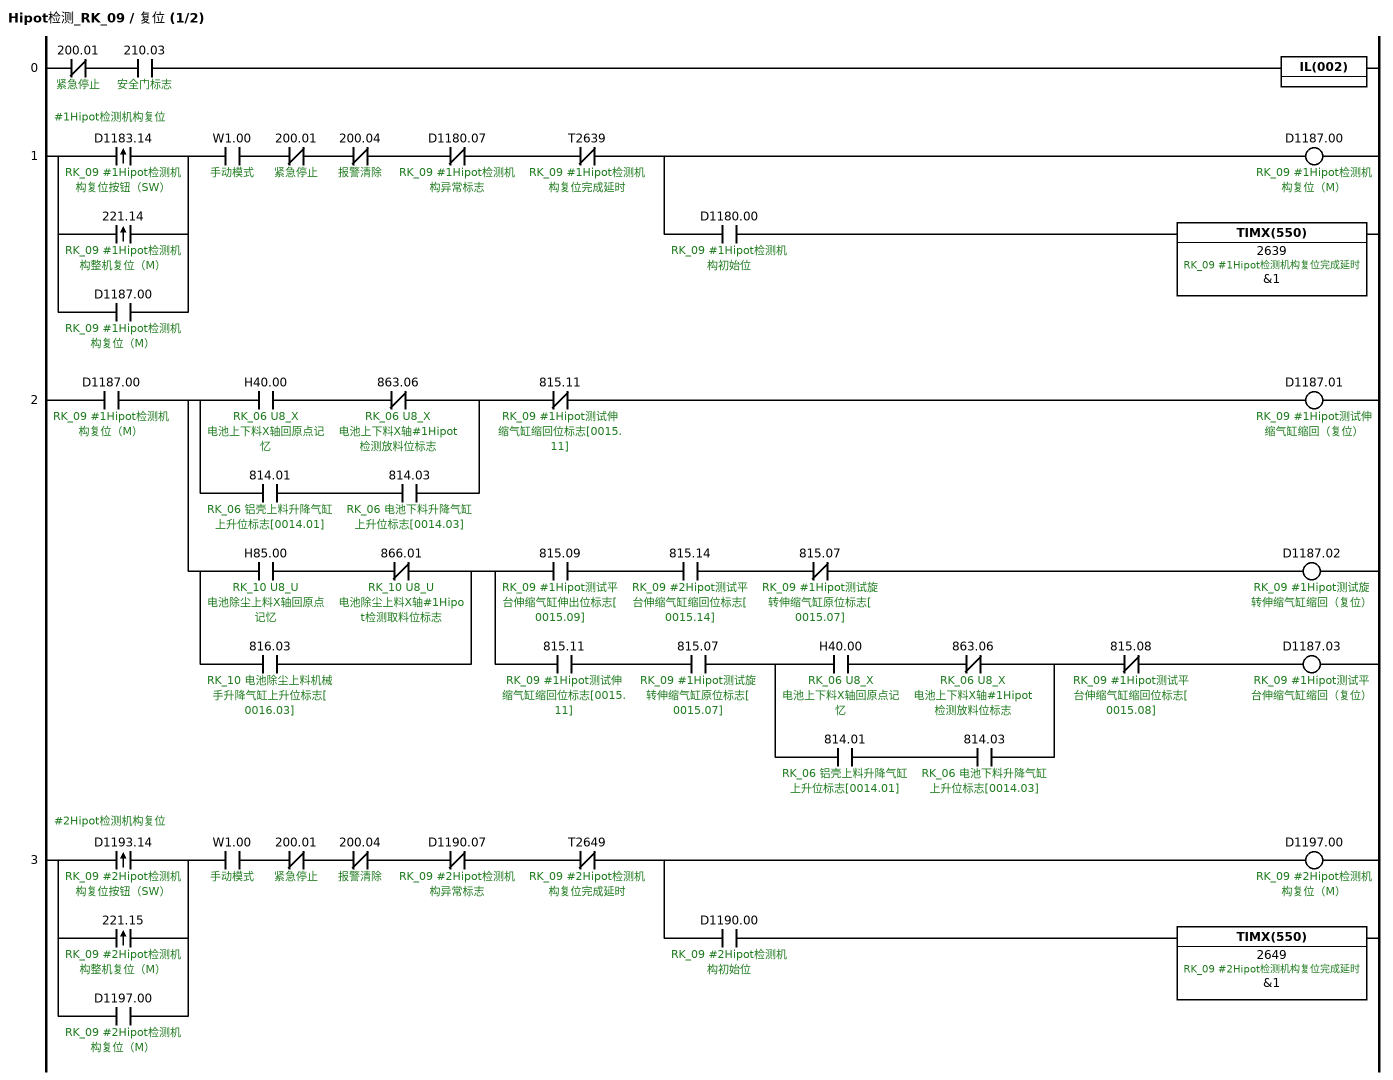
; [picture p672: Hipot检测_RK_09 / 复位, rungs 0-3]
; rung 0
LDNOT 200.01  ; 紧急停止
AND 210.03  ; 安全门标志
IL(002)
; rung 1: #1Hipot检测机构复位
@LD D1183.14  ; RK_09 #1Hipot检测机构复位按钮（SW）
@OR 221.14  ; RK_09 #1Hipot检测机构整机复位（M）
OR D1187.00  ; RK_09 #1Hipot检测机构复位（M）
AND W1.00  ; 手动模式
ANDNOT 200.01  ; 紧急停止
ANDNOT 200.04  ; 报警清除
ANDNOT D1180.07  ; RK_09 #1Hipot检测机构异常标志
ANDNOT T2639  ; RK_09 #1Hipot检测机构复位完成延时
OUT D1187.00  ; RK_09 #1Hipot检测机构复位（M）
AND D1180.00  ; RK_09 #1Hipot检测机构初始位
TIMX(550) 2639 &1  ; RK_09 #1Hipot检测机构复位完成延时
; rung 2
LD D1187.00  ; RK_09 #1Hipot检测机构复位（M）
OUT TR0
LD H40.00  ; RK_06 U8_X 电池上下料X轴回原点记忆
ANDNOT 863.06  ; RK_06 U8_X 电池上下料X轴#1Hipot检测放料位标志
LD 814.01  ; RK_06 铝壳上料升降气缸上升位标志[0014.01]
AND 814.03  ; RK_06 电池下料升降气缸上升位标志[0014.03]
ORLD
ANDLD
ANDNOT 815.11  ; RK_09 #1Hipot测试伸缩气缸缩回位标志[0015.11]
OUT D1187.01  ; RK_09 #1Hipot测试伸缩气缸缩回（复位）
LD TR0
LD H85.00  ; RK_10 U8_U 电池除尘上料X轴回原点记忆
ANDNOT 866.01  ; RK_10 U8_U 电池除尘上料X轴#1Hipot检测取料位标志
OR 816.03  ; RK_10 电池除尘上料机械手升降气缸上升位标志[0016.03]
ANDLD
OUT TR0
AND 815.09  ; RK_09 #1Hipot测试平台伸缩气缸伸出位标志[0015.09]
AND 815.14  ; RK_09 #2Hipot测试平台伸缩气缸缩回位标志[0015.14]
ANDNOT 815.07  ; RK_09 #1Hipot测试旋转伸缩气缸原位标志[0015.07]
OUT D1187.02  ; RK_09 #1Hipot测试旋转伸缩气缸缩回（复位）
LD TR0
AND 815.11  ; RK_09 #1Hipot测试伸缩气缸缩回位标志[0015.11]
AND 815.07  ; RK_09 #1Hipot测试旋转伸缩气缸原位标志[0015.07]
LD H40.00  ; RK_06 U8_X 电池上下料X轴回原点记忆
ANDNOT 863.06  ; RK_06 U8_X 电池上下料X轴#1Hipot检测放料位标志
LD 814.01  ; RK_06 铝壳上料升降气缸上升位标志[0014.01]
AND 814.03  ; RK_06 电池下料升降气缸上升位标志[0014.03]
ORLD
ANDLD
ANDNOT 815.08  ; RK_09 #1Hipot测试平台伸缩气缸缩回位标志[0015.08]
OUT D1187.03  ; RK_09 #1Hipot测试平台伸缩气缸缩回（复位）
; rung 3: #2Hipot检测机构复位
@LD D1193.14  ; RK_09 #2Hipot检测机构复位按钮（SW）
@OR 221.15  ; RK_09 #2Hipot检测机构整机复位（M）
OR D1197.00  ; RK_09 #2Hipot检测机构复位（M）
AND W1.00  ; 手动模式
ANDNOT 200.01  ; 紧急停止
ANDNOT 200.04  ; 报警清除
ANDNOT D1190.07  ; RK_09 #2Hipot检测机构异常标志
ANDNOT T2649  ; RK_09 #2Hipot检测机构复位完成延时
OUT D1197.00  ; RK_09 #2Hipot检测机构复位（M）
AND D1190.00  ; RK_09 #2Hipot检测机构初始位
TIMX(550) 2649 &1  ; RK_09 #2Hipot检测机构复位完成延时

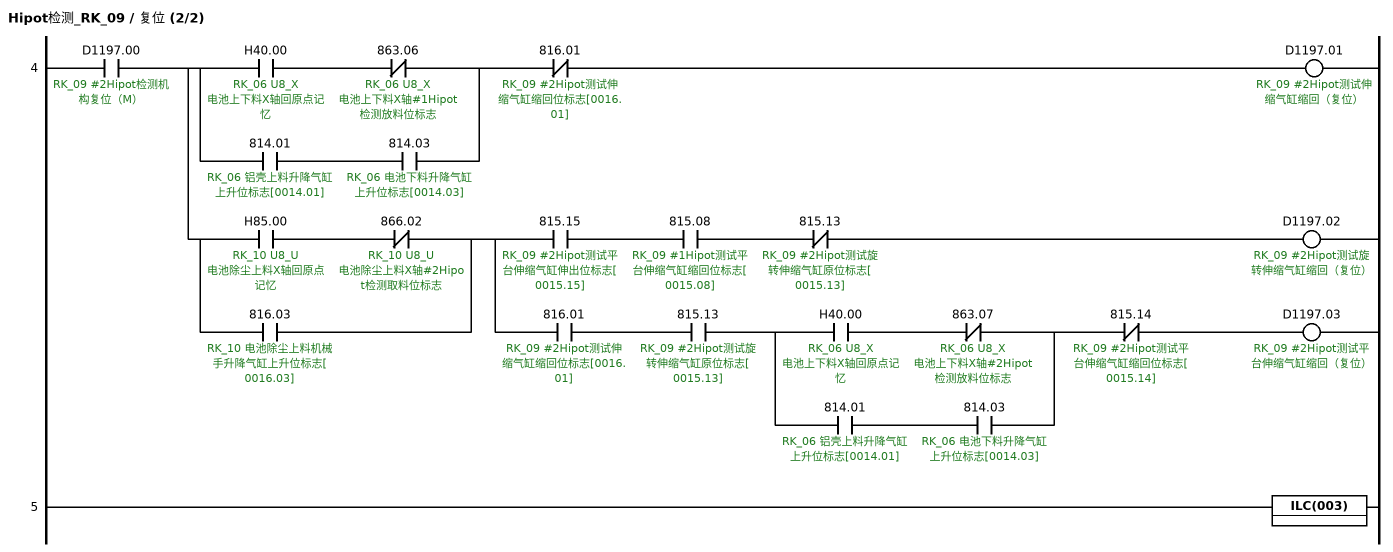
; rung 4
LD D1197.00  ; RK_09 #2Hipot检测机构复位（M）
OUT TR0
LD H40.00  ; RK_06 U8_X 电池上下料X轴回原点记忆
ANDNOT 863.06  ; RK_06 U8_X 电池上下料X轴#1Hipot检测放料位标志
LD 814.01  ; RK_06 铝壳上料升降气缸上升位标志[0014.01]
AND 814.03  ; RK_06 电池下料升降气缸上升位标志[0014.03]
ORLD
ANDLD
ANDNOT 816.01  ; RK_09 #2Hipot测试伸缩气缸缩回位标志[0016.01]
OUT D1197.01  ; RK_09 #2Hipot测试伸缩气缸缩回（复位）
LD TR0
LD H85.00  ; RK_10 U8_U 电池除尘上料X轴回原点记忆
ANDNOT 866.02  ; RK_10 U8_U 电池除尘上料X轴#2Hipot检测取料位标志
OR 816.03  ; RK_10 电池除尘上料机械手升降气缸上升位标志[0016.03]
ANDLD
OUT TR0
AND 815.15  ; RK_09 #2Hipot测试平台伸缩气缸伸出位标志[0015.15]
AND 815.08  ; RK_09 #1Hipot测试平台伸缩气缸缩回位标志[0015.08]
ANDNOT 815.13  ; RK_09 #2Hipot测试旋转伸缩气缸原位标志[0015.13]
OUT D1197.02  ; RK_09 #2Hipot测试旋转伸缩气缸缩回（复位）
LD TR0
AND 816.01  ; RK_09 #2Hipot测试伸缩气缸缩回位标志[0016.01]
AND 815.13  ; RK_09 #2Hipot测试旋转伸缩气缸原位标志[0015.13]
LD H40.00  ; RK_06 U8_X 电池上下料X轴回原点记忆
ANDNOT 863.07  ; RK_06 U8_X 电池上下料X轴#2Hipot检测放料位标志
LD 814.01  ; RK_06 铝壳上料升降气缸上升位标志[0014.01]
AND 814.03  ; RK_06 电池下料升降气缸上升位标志[0014.03]
ORLD
ANDLD
ANDNOT 815.14  ; RK_09 #2Hipot测试平台伸缩气缸缩回位标志[0015.14]
OUT D1197.03  ; RK_09 #2Hipot测试平台伸缩气缸缩回（复位）
; rung 5
ILC(003)

### Section 指示灯

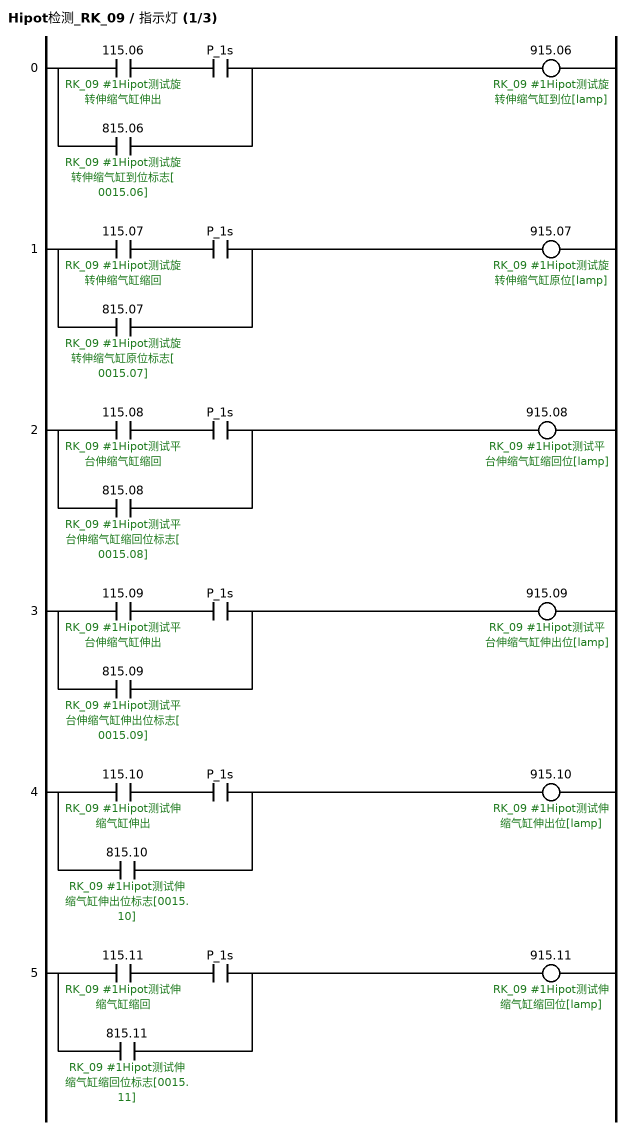
; rung 0
LD 115.06  ; RK_09 #1Hipot测试旋转伸缩气缸伸出
AND P_1s
OR 815.06  ; RK_09 #1Hipot测试旋转伸缩气缸到位标志[0015.06]
OUT 915.06  ; RK_09 #1Hipot测试旋转伸缩气缸到位[lamp]
; rung 1
LD 115.07  ; RK_09 #1Hipot测试旋转伸缩气缸缩回
AND P_1s
OR 815.07  ; RK_09 #1Hipot测试旋转伸缩气缸原位标志[0015.07]
OUT 915.07  ; RK_09 #1Hipot测试旋转伸缩气缸原位[lamp]
; rung 2
LD 115.08  ; RK_09 #1Hipot测试平台伸缩气缸缩回
AND P_1s
OR 815.08  ; RK_09 #1Hipot测试平台伸缩气缸缩回位标志[0015.08]
OUT 915.08  ; RK_09 #1Hipot测试平台伸缩气缸缩回位[lamp]
; rung 3
LD 115.09  ; RK_09 #1Hipot测试平台伸缩气缸伸出
AND P_1s
OR 815.09  ; RK_09 #1Hipot测试平台伸缩气缸伸出位标志[0015.09]
OUT 915.09  ; RK_09 #1Hipot测试平台伸缩气缸伸出位[lamp]
; rung 4
LD 115.10  ; RK_09 #1Hipot测试伸缩气缸伸出
AND P_1s
OR 815.10  ; RK_09 #1Hipot测试伸缩气缸伸出位标志[0015.10]
OUT 915.10  ; RK_09 #1Hipot测试伸缩气缸伸出位[lamp]
; rung 5
LD 115.11  ; RK_09 #1Hipot测试伸缩气缸缩回
AND P_1s
OR 815.11  ; RK_09 #1Hipot测试伸缩气缸缩回位标志[0015.11]
OUT 915.11  ; RK_09 #1Hipot测试伸缩气缸缩回位[lamp]

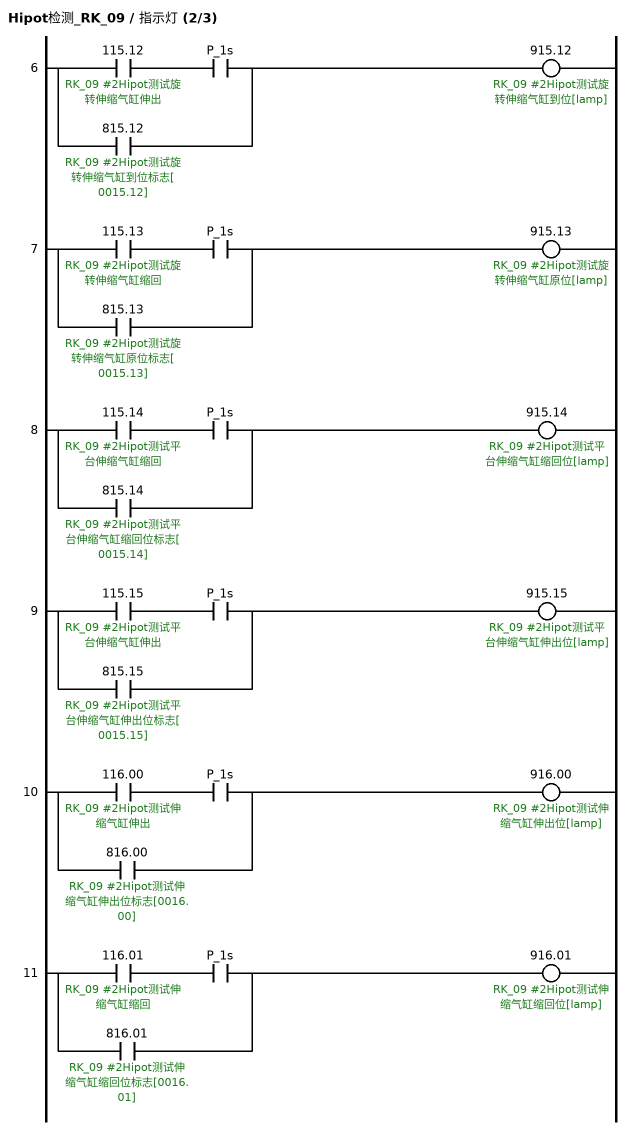
; rung 6
LD 115.12  ; RK_09 #2Hipot测试旋转伸缩气缸伸出
AND P_1s
OR 815.12  ; RK_09 #2Hipot测试旋转伸缩气缸到位标志[0015.12]
OUT 915.12  ; RK_09 #2Hipot测试旋转伸缩气缸到位[lamp]
; rung 7
LD 115.13  ; RK_09 #2Hipot测试旋转伸缩气缸缩回
AND P_1s
OR 815.13  ; RK_09 #2Hipot测试旋转伸缩气缸原位标志[0015.13]
OUT 915.13  ; RK_09 #2Hipot测试旋转伸缩气缸原位[lamp]
; rung 8
LD 115.14  ; RK_09 #2Hipot测试平台伸缩气缸缩回
AND P_1s
OR 815.14  ; RK_09 #2Hipot测试平台伸缩气缸缩回位标志[0015.14]
OUT 915.14  ; RK_09 #2Hipot测试平台伸缩气缸缩回位[lamp]
; rung 9
LD 115.15  ; RK_09 #2Hipot测试平台伸缩气缸伸出
AND P_1s
OR 815.15  ; RK_09 #2Hipot测试平台伸缩气缸伸出位标志[0015.15]
OUT 915.15  ; RK_09 #2Hipot测试平台伸缩气缸伸出位[lamp]
; rung 10
LD 116.00  ; RK_09 #2Hipot测试伸缩气缸伸出
AND P_1s
OR 816.00  ; RK_09 #2Hipot测试伸缩气缸伸出位标志[0016.00]
OUT 916.00  ; RK_09 #2Hipot测试伸缩气缸伸出位[lamp]
; rung 11
LD 116.01  ; RK_09 #2Hipot测试伸缩气缸缩回
AND P_1s
OR 816.01  ; RK_09 #2Hipot测试伸缩气缸缩回位标志[0016.01]
OUT 916.01  ; RK_09 #2Hipot测试伸缩气缸缩回位[lamp]

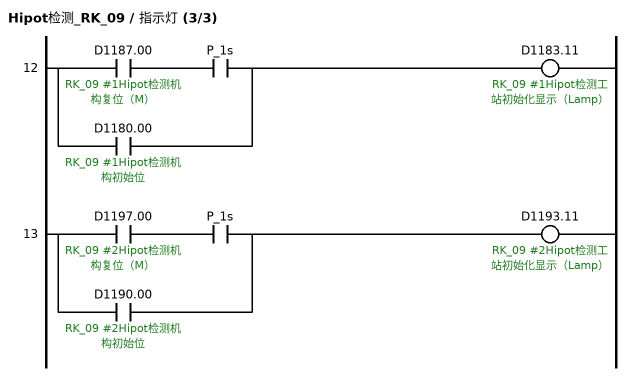
; rung 12
LD D1187.00  ; RK_09 #1Hipot检测机构复位（M）
AND P_1s
OR D1180.00  ; RK_09 #1Hipot检测机构初始位
OUT D1183.11  ; RK_09 #1Hipot检测工站初始化显示（Lamp）
; rung 13
LD D1197.00  ; RK_09 #2Hipot检测机构复位（M）
AND P_1s
OR D1190.00  ; RK_09 #2Hipot检测机构初始位
OUT D1193.11  ; RK_09 #2Hipot检测工站初始化显示（Lamp）

### Section 外部输出

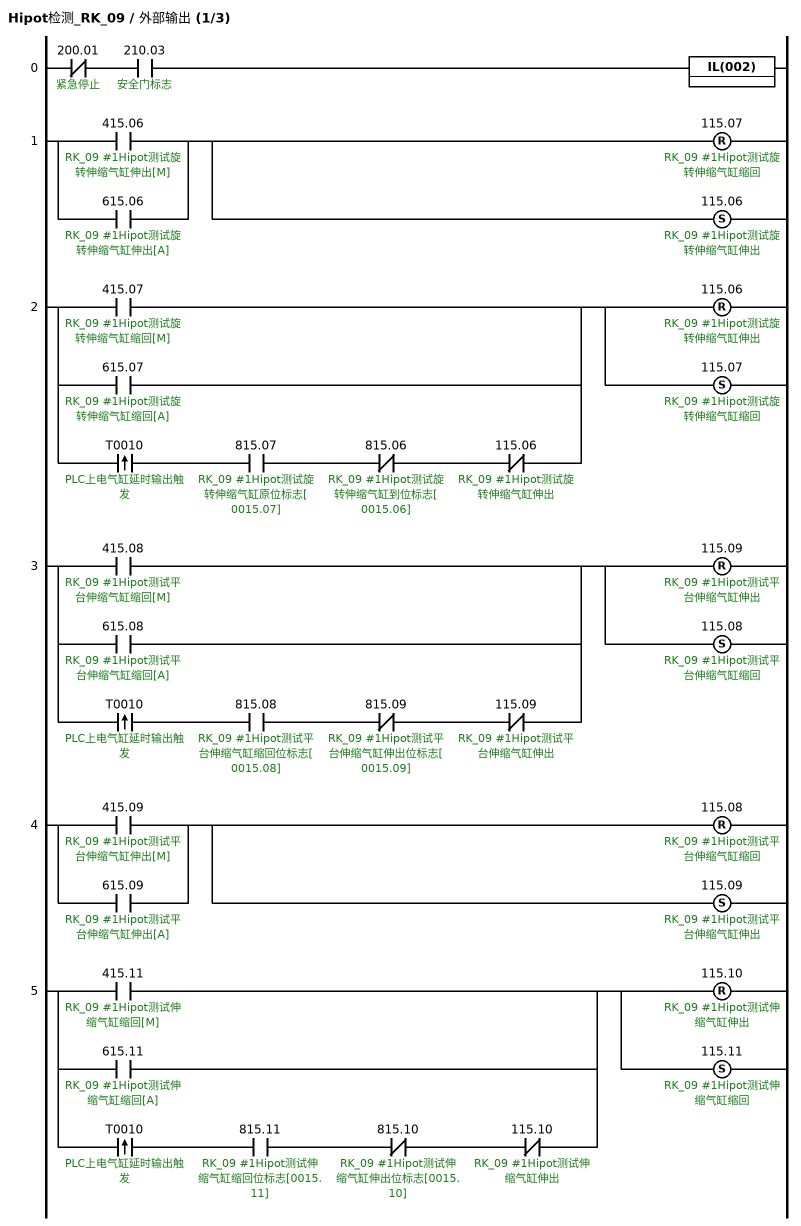
; rung 0
LDNOT 200.01  ; 紧急停止
AND 210.03  ; 安全门标志
IL(002)
; rung 1
LD 415.06  ; RK_09 #1Hipot测试旋转伸缩气缸伸出[M]
OR 615.06  ; RK_09 #1Hipot测试旋转伸缩气缸伸出[A]
RSET 115.07  ; RK_09 #1Hipot测试旋转伸缩气缸缩回
SET 115.06  ; RK_09 #1Hipot测试旋转伸缩气缸伸出
; rung 2
LD 415.07  ; RK_09 #1Hipot测试旋转伸缩气缸缩回[M]
OR 615.07  ; RK_09 #1Hipot测试旋转伸缩气缸缩回[A]
@LD T0010  ; PLC上电气缸延时输出触发
AND 815.07  ; RK_09 #1Hipot测试旋转伸缩气缸原位标志[0015.07]
ANDNOT 815.06  ; RK_09 #1Hipot测试旋转伸缩气缸到位标志[0015.06]
ANDNOT 115.06  ; RK_09 #1Hipot测试旋转伸缩气缸伸出
ORLD
RSET 115.06  ; RK_09 #1Hipot测试旋转伸缩气缸伸出
SET 115.07  ; RK_09 #1Hipot测试旋转伸缩气缸缩回
; rung 3
LD 415.08  ; RK_09 #1Hipot测试平台伸缩气缸缩回[M]
OR 615.08  ; RK_09 #1Hipot测试平台伸缩气缸缩回[A]
@LD T0010  ; PLC上电气缸延时输出触发
AND 815.08  ; RK_09 #1Hipot测试平台伸缩气缸缩回位标志[0015.08]
ANDNOT 815.09  ; RK_09 #1Hipot测试平台伸缩气缸伸出位标志[0015.09]
ANDNOT 115.09  ; RK_09 #1Hipot测试平台伸缩气缸伸出
ORLD
RSET 115.09  ; RK_09 #1Hipot测试平台伸缩气缸伸出
SET 115.08  ; RK_09 #1Hipot测试平台伸缩气缸缩回
; rung 4
LD 415.09  ; RK_09 #1Hipot测试平台伸缩气缸伸出[M]
OR 615.09  ; RK_09 #1Hipot测试平台伸缩气缸伸出[A]
RSET 115.08  ; RK_09 #1Hipot测试平台伸缩气缸缩回
SET 115.09  ; RK_09 #1Hipot测试平台伸缩气缸伸出
; rung 5
LD 415.11  ; RK_09 #1Hipot测试伸缩气缸缩回[M]
OR 615.11  ; RK_09 #1Hipot测试伸缩气缸缩回[A]
@LD T0010  ; PLC上电气缸延时输出触发
AND 815.11  ; RK_09 #1Hipot测试伸缩气缸缩回位标志[0015.11]
ANDNOT 815.10  ; RK_09 #1Hipot测试伸缩气缸伸出位标志[0015.10]
ANDNOT 115.10  ; RK_09 #1Hipot测试伸缩气缸伸出
ORLD
RSET 115.10  ; RK_09 #1Hipot测试伸缩气缸伸出
SET 115.11  ; RK_09 #1Hipot测试伸缩气缸缩回

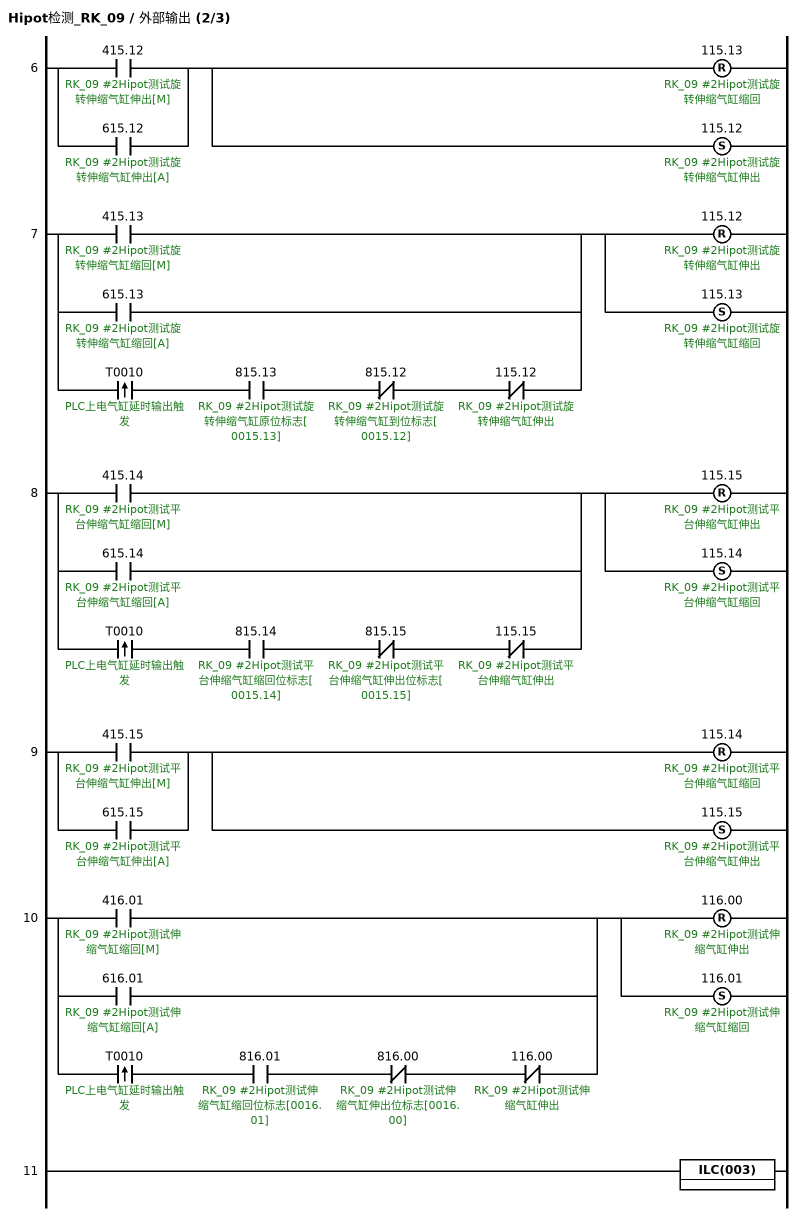
; rung 6
LD 415.12  ; RK_09 #2Hipot测试旋转伸缩气缸伸出[M]
OR 615.12  ; RK_09 #2Hipot测试旋转伸缩气缸伸出[A]
RSET 115.13  ; RK_09 #2Hipot测试旋转伸缩气缸缩回
SET 115.12  ; RK_09 #2Hipot测试旋转伸缩气缸伸出
; rung 7
LD 415.13  ; RK_09 #2Hipot测试旋转伸缩气缸缩回[M]
OR 615.13  ; RK_09 #2Hipot测试旋转伸缩气缸缩回[A]
@LD T0010  ; PLC上电气缸延时输出触发
AND 815.13  ; RK_09 #2Hipot测试旋转伸缩气缸原位标志[0015.13]
ANDNOT 815.12  ; RK_09 #2Hipot测试旋转伸缩气缸到位标志[0015.12]
ANDNOT 115.12  ; RK_09 #2Hipot测试旋转伸缩气缸伸出
ORLD
RSET 115.12  ; RK_09 #2Hipot测试旋转伸缩气缸伸出
SET 115.13  ; RK_09 #2Hipot测试旋转伸缩气缸缩回
; rung 8
LD 415.14  ; RK_09 #2Hipot测试平台伸缩气缸缩回[M]
OR 615.14  ; RK_09 #2Hipot测试平台伸缩气缸缩回[A]
@LD T0010  ; PLC上电气缸延时输出触发
AND 815.14  ; RK_09 #2Hipot测试平台伸缩气缸缩回位标志[0015.14]
ANDNOT 815.15  ; RK_09 #2Hipot测试平台伸缩气缸伸出位标志[0015.15]
ANDNOT 115.15  ; RK_09 #2Hipot测试平台伸缩气缸伸出
ORLD
RSET 115.15  ; RK_09 #2Hipot测试平台伸缩气缸伸出
SET 115.14  ; RK_09 #2Hipot测试平台伸缩气缸缩回
; rung 9
LD 415.15  ; RK_09 #2Hipot测试平台伸缩气缸伸出[M]
OR 615.15  ; RK_09 #2Hipot测试平台伸缩气缸伸出[A]
RSET 115.14  ; RK_09 #2Hipot测试平台伸缩气缸缩回
SET 115.15  ; RK_09 #2Hipot测试平台伸缩气缸伸出
; rung 10
LD 416.01  ; RK_09 #2Hipot测试伸缩气缸缩回[M]
OR 616.01  ; RK_09 #2Hipot测试伸缩气缸缩回[A]
@LD T0010  ; PLC上电气缸延时输出触发
AND 816.01  ; RK_09 #2Hipot测试伸缩气缸缩回位标志[0016.01]
ANDNOT 816.00  ; RK_09 #2Hipot测试伸缩气缸伸出位标志[0016.00]
ANDNOT 116.00  ; RK_09 #2Hipot测试伸缩气缸伸出
ORLD
RSET 116.00  ; RK_09 #2Hipot测试伸缩气缸伸出
SET 116.01  ; RK_09 #2Hipot测试伸缩气缸缩回
; rung 11
ILC(003)

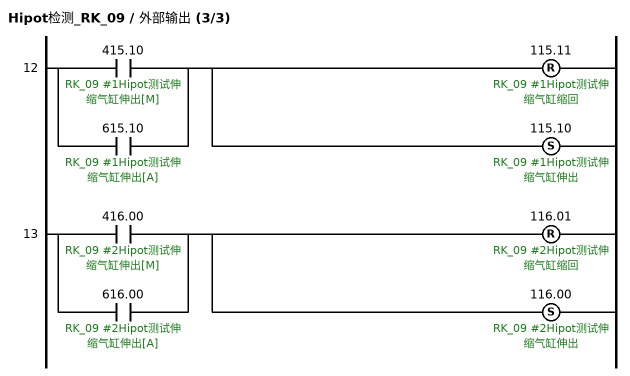
; rung 12
LD 415.10  ; RK_09 #1Hipot测试伸缩气缸伸出[M]
OR 615.10  ; RK_09 #1Hipot测试伸缩气缸伸出[A]
RSET 115.11  ; RK_09 #1Hipot测试伸缩气缸缩回
SET 115.10  ; RK_09 #1Hipot测试伸缩气缸伸出
; rung 13
LD 416.00  ; RK_09 #2Hipot测试伸缩气缸伸出[M]
OR 616.00  ; RK_09 #2Hipot测试伸缩气缸伸出[A]
RSET 116.01  ; RK_09 #2Hipot测试伸缩气缸缩回
SET 116.00  ; RK_09 #2Hipot测试伸缩气缸伸出

### Section END
; rung 0
END(001)

## Program 电池除尘上料_RK_10 (cyclic task 10)

### Section Main

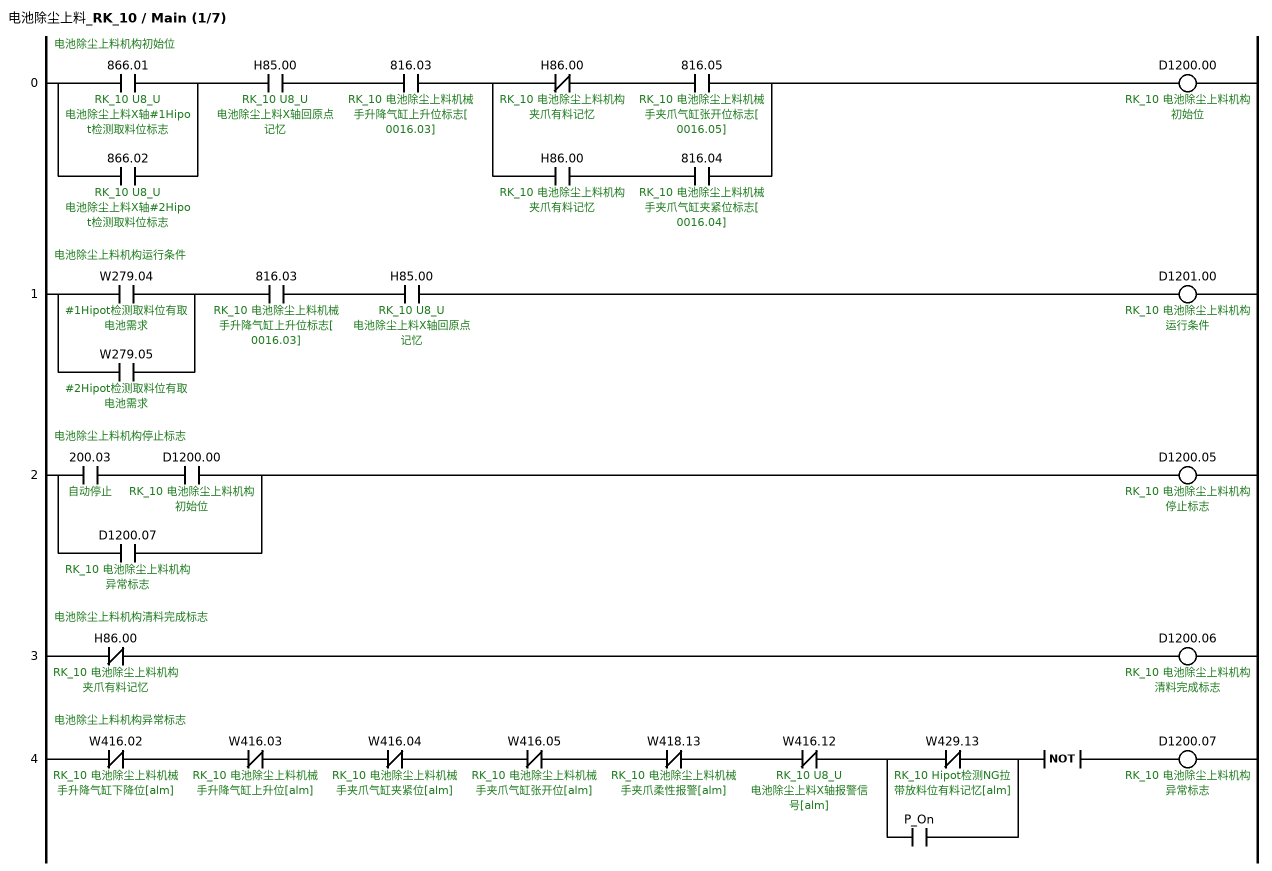
; rung 0: 电池除尘上料机构初始位
LD 866.01  ; RK_10 U8_U 电池除尘上料X轴#1Hipot检测取料位标志
OR 866.02  ; RK_10 U8_U 电池除尘上料X轴#2Hipot检测取料位标志
AND H85.00  ; RK_10 U8_U 电池除尘上料X轴回原点记忆
AND 816.03  ; RK_10 电池除尘上料机械手升降气缸上升位标志[0016.03]
LDNOT H86.00  ; RK_10 电池除尘上料机构夹爪有料记忆
AND 816.05  ; RK_10 电池除尘上料机械手夹爪气缸张开位标志[0016.05]
LD H86.00  ; RK_10 电池除尘上料机构夹爪有料记忆
AND 816.04  ; RK_10 电池除尘上料机械手夹爪气缸夹紧位标志[0016.04]
ORLD
ANDLD
OUT D1200.00  ; RK_10 电池除尘上料机构初始位
; rung 1: 电池除尘上料机构运行条件
LD W279.04  ; #1Hipot检测取料位有取电池需求
OR W279.05  ; #2Hipot检测取料位有取电池需求
AND 816.03  ; RK_10 电池除尘上料机械手升降气缸上升位标志[0016.03]
AND H85.00  ; RK_10 U8_U 电池除尘上料X轴回原点记忆
OUT D1201.00  ; RK_10 电池除尘上料机构运行条件
; rung 2: 电池除尘上料机构停止标志
LD 200.03  ; 自动停止
AND D1200.00  ; RK_10 电池除尘上料机构初始位
OR D1200.07  ; RK_10 电池除尘上料机构异常标志
OUT D1200.05  ; RK_10 电池除尘上料机构停止标志
; rung 3: 电池除尘上料机构清料完成标志
LDNOT H86.00  ; RK_10 电池除尘上料机构夹爪有料记忆
OUT D1200.06  ; RK_10 电池除尘上料机构清料完成标志
; rung 4: 电池除尘上料机构异常标志
LDNOT W416.02  ; RK_10 电池除尘上料机械手升降气缸下降位[alm]
ANDNOT W416.03  ; RK_10 电池除尘上料机械手升降气缸上升位[alm]
ANDNOT W416.04  ; RK_10 电池除尘上料机械手夹爪气缸夹紧位[alm]
ANDNOT W416.05  ; RK_10 电池除尘上料机械手夹爪气缸张开位[alm]
ANDNOT W418.13  ; RK_10 电池除尘上料机械手夹爪柔性报警[alm]
ANDNOT W416.12  ; RK_10 U8_U 电池除尘上料X轴报警信号[alm]
LDNOT W429.13  ; RK_10 Hipot检测NG拉带放料位有料记忆[alm]
OR P_On
ANDLD
NOT(520)
OUT D1200.07  ; RK_10 电池除尘上料机构异常标志

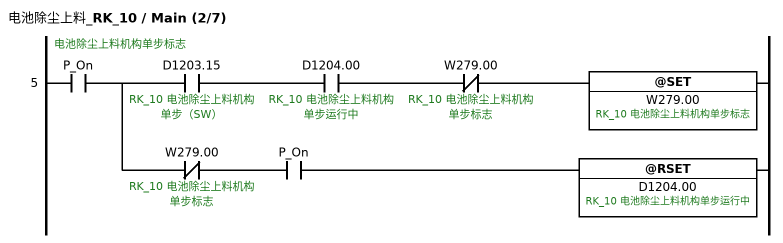
; rung 5: 电池除尘上料机构单步标志
LD P_On
OUT TR0
AND D1203.15  ; RK_10 电池除尘上料机构单步（SW）
AND D1204.00  ; RK_10 电池除尘上料机构单步运行中
ANDNOT W279.00  ; RK_10 电池除尘上料机构单步标志
@SET W279.00  ; RK_10 电池除尘上料机构单步标志
LD TR0
ANDNOT W279.00  ; RK_10 电池除尘上料机构单步标志
AND P_On
@RSET D1204.00  ; RK_10 电池除尘上料机构单步运行中

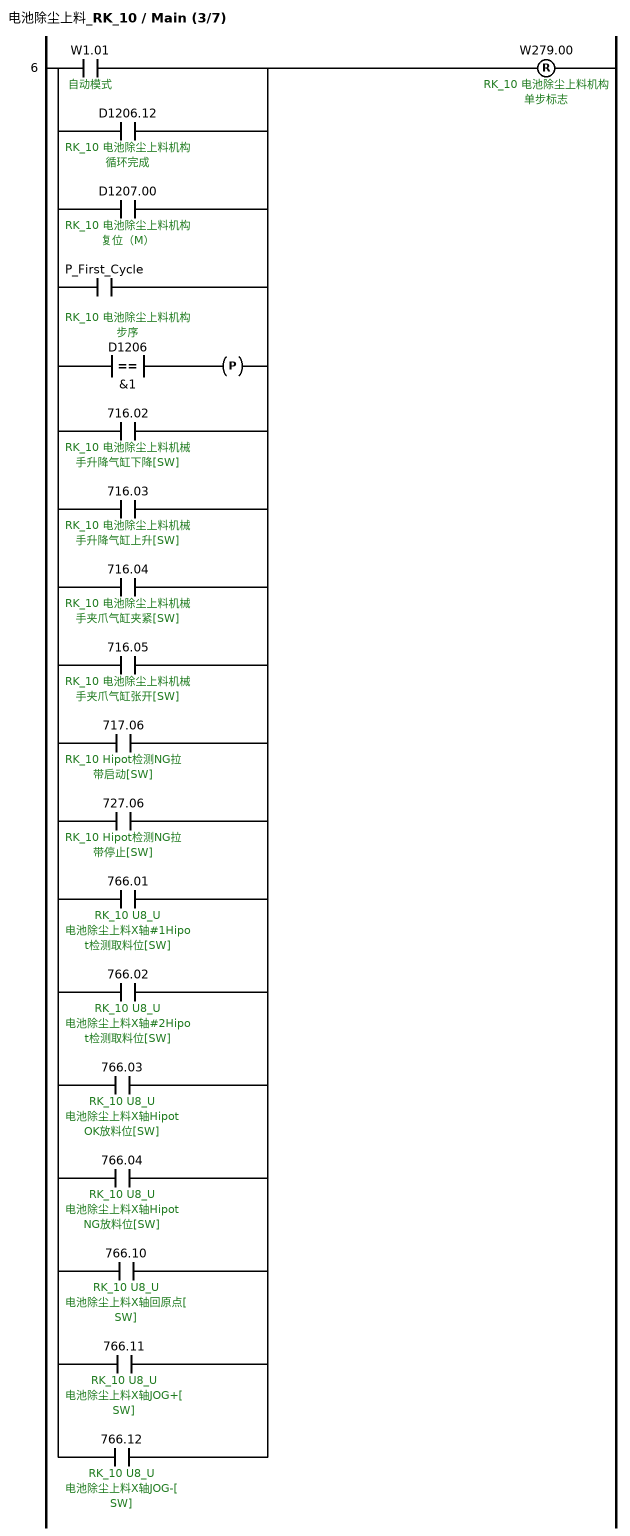
; rung 6
LD W1.01  ; 自动模式
OR D1206.12  ; RK_10 电池除尘上料机构循环完成
OR D1207.00  ; RK_10 电池除尘上料机构复位（M）
OR P_First_Cycle
LD=(300) D1206 &1  ; RK_10 电池除尘上料机构步序
UP(521)
ORLD
LD 716.02  ; RK_10 电池除尘上料机械手升降气缸下降[SW]
OR 716.03  ; RK_10 电池除尘上料机械手升降气缸上升[SW]
OR 716.04  ; RK_10 电池除尘上料机械手夹爪气缸夹紧[SW]
OR 716.05  ; RK_10 电池除尘上料机械手夹爪气缸张开[SW]
OR 717.06  ; RK_10 Hipot检测NG拉带启动[SW]
OR 727.06  ; RK_10 Hipot检测NG拉带停止[SW]
OR 766.01  ; RK_10 U8_U 电池除尘上料X轴#1Hipot检测取料位[SW]
OR 766.02  ; RK_10 U8_U 电池除尘上料X轴#2Hipot检测取料位[SW]
OR 766.03  ; RK_10 U8_U 电池除尘上料X轴Hipot OK放料位[SW]
OR 766.04  ; RK_10 U8_U 电池除尘上料X轴Hipot NG放料位[SW]
OR 766.10  ; RK_10 U8_U 电池除尘上料X轴回原点[SW]
OR 766.11  ; RK_10 U8_U 电池除尘上料X轴JOG+[SW]
OR 766.12  ; RK_10 U8_U 电池除尘上料X轴JOG-[SW]
ORLD
RSET W279.00  ; RK_10 电池除尘上料机构单步标志

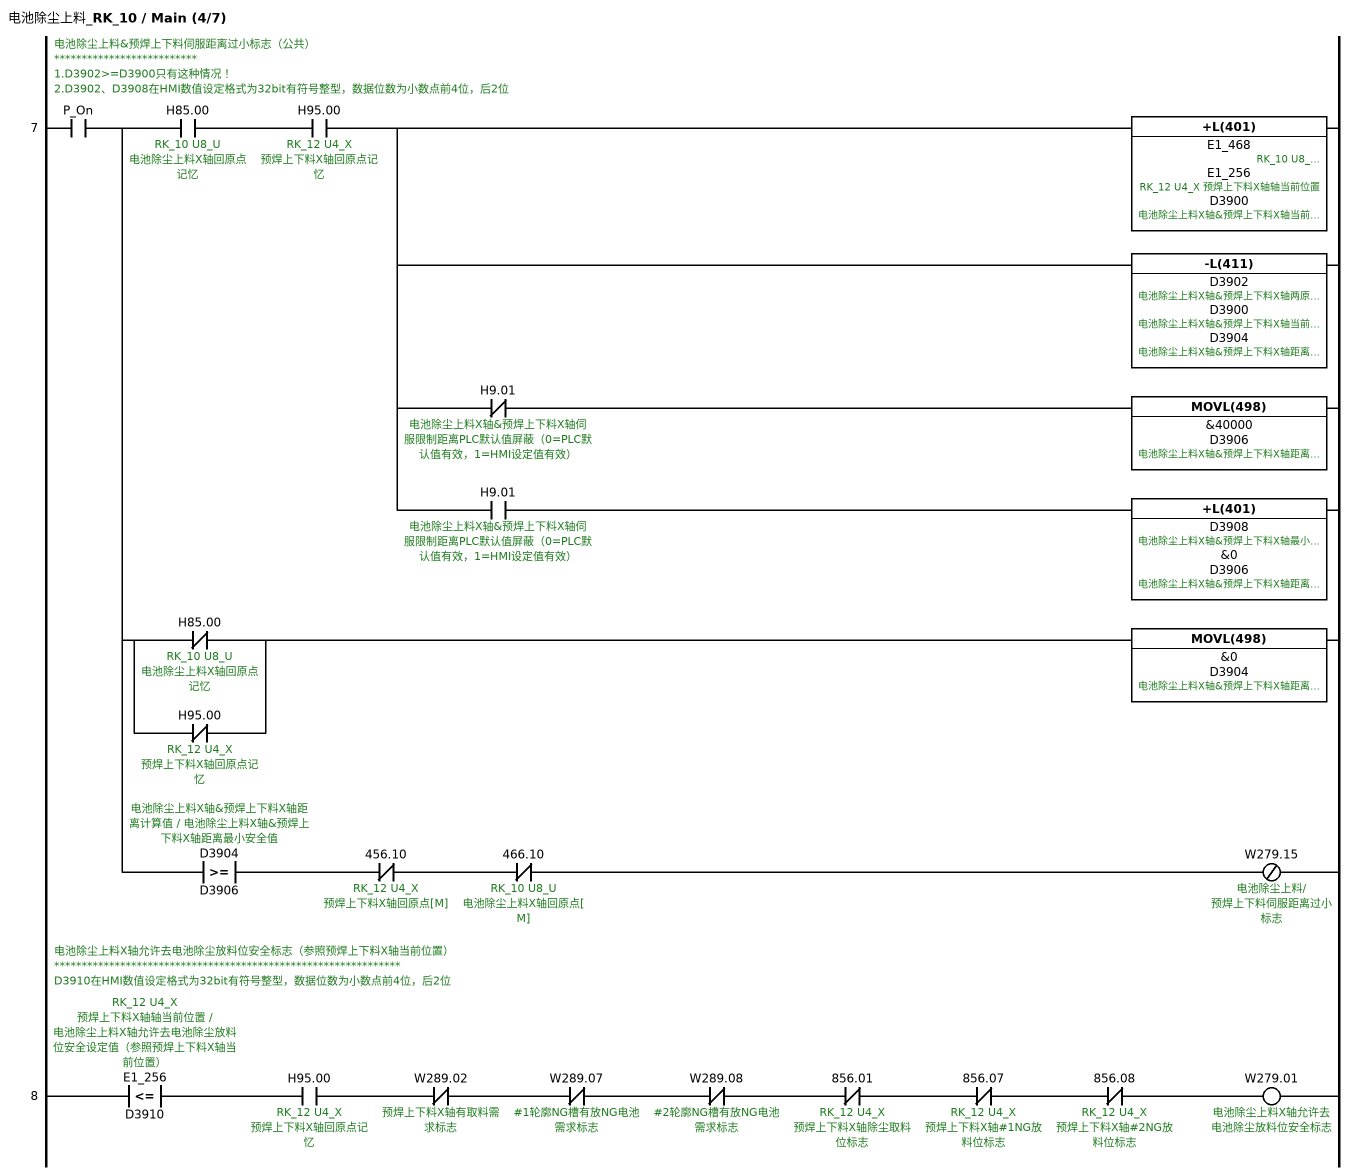
; rung 7: 电池除尘上料&预焊上下料伺服距离过小标志（公共） / ************************** / 1.D3902>=D3900只有这种情况！ / 2.D3902、D3908在HMI数值设定格式为32bit有符号整型，数据位数为小数点前4位，后2位
LD P_On
OUT TR0
AND H85.00  ; RK_10 U8_U 电池除尘上料X轴回原点记忆
AND H95.00  ; RK_12 U4_X 预焊上下料X轴回原点记忆
OUT TR1
+L(401) E1_468 E1_256 D3900  ; RK_10 U8_U 电池除尘上料X轴轴当前位置, RK_12 U4_X 预焊上下料X轴轴当前位置, 电池除尘上料X轴&预焊上下料X轴当前总距离
-L(411) D3902 D3900 D3904  ; 电池除尘上料X轴&预焊上下料X轴两原点间距离设定值, 电池除尘上料X轴&预焊上下料X轴当前总距离, 电池除尘上料X轴&预焊上下料X轴距离计算值
ANDNOT H9.01  ; 电池除尘上料X轴&预焊上下料X轴伺服限制距离PLC默认值屏蔽（0=PLC默认值有效，1=HMI设定值有效）
MOVL(498) &40000 D3906  ; 电池除尘上料X轴&预焊上下料X轴距离最小安全值
LD TR1
AND H9.01  ; 电池除尘上料X轴&预焊上下料X轴伺服限制距离PLC默认值屏蔽（0=PLC默认值有效，1=HMI设定值有效）
+L(401) D3908 &0 D3906  ; 电池除尘上料X轴&预焊上下料X轴最小安全距离设定值, 电池除尘上料X轴&预焊上下料X轴距离最小安全值
LD TR0
LDNOT H85.00  ; RK_10 U8_U 电池除尘上料X轴回原点记忆
ORNOT H95.00  ; RK_12 U4_X 预焊上下料X轴回原点记忆
ANDLD
MOVL(498) &0 D3904  ; 电池除尘上料X轴&预焊上下料X轴距离计算值
LD TR0
AND>=SL(328) D3904 D3906  ; 电池除尘上料X轴&预焊上下料X轴距离计算值, 电池除尘上料X轴&预焊上下料X轴距离最小安全值
ANDNOT 456.10  ; RK_12 U4_X 预焊上下料X轴回原点[M]
ANDNOT 466.10  ; RK_10 U8_U 电池除尘上料X轴回原点[M]
OUTNOT W279.15  ; 电池除尘上料/预焊上下料伺服距离过小标志
; rung 8: 电池除尘上料X轴允许去电池除尘放料位安全标志（参照预焊上下料X轴当前位置） / *************************************************************** / D3910在HMI数值设定格式为32bit有符号整型，数据位数为小数点前4位，后2位
LD<=SL(318) E1_256 D3910  ; RK_12 U4_X 预焊上下料X轴轴当前位置, 电池除尘上料X轴允许去电池除尘放料位安全设定值（参照预焊上下料X轴当前位置）
AND H95.00  ; RK_12 U4_X 预焊上下料X轴回原点记忆
ANDNOT W289.02  ; 预焊上下料X轴有取料需求标志
ANDNOT W289.07  ; #1轮廓NG槽有放NG电池需求标志
ANDNOT W289.08  ; #2轮廓NG槽有放NG电池需求标志
ANDNOT 856.01  ; RK_12 U4_X 预焊上下料X轴除尘取料位标志
ANDNOT 856.07  ; RK_12 U4_X 预焊上下料X轴#1NG放料位标志
ANDNOT 856.08  ; RK_12 U4_X 预焊上下料X轴#2NG放料位标志
OUT W279.01  ; 电池除尘上料X轴允许去电池除尘放料位安全标志

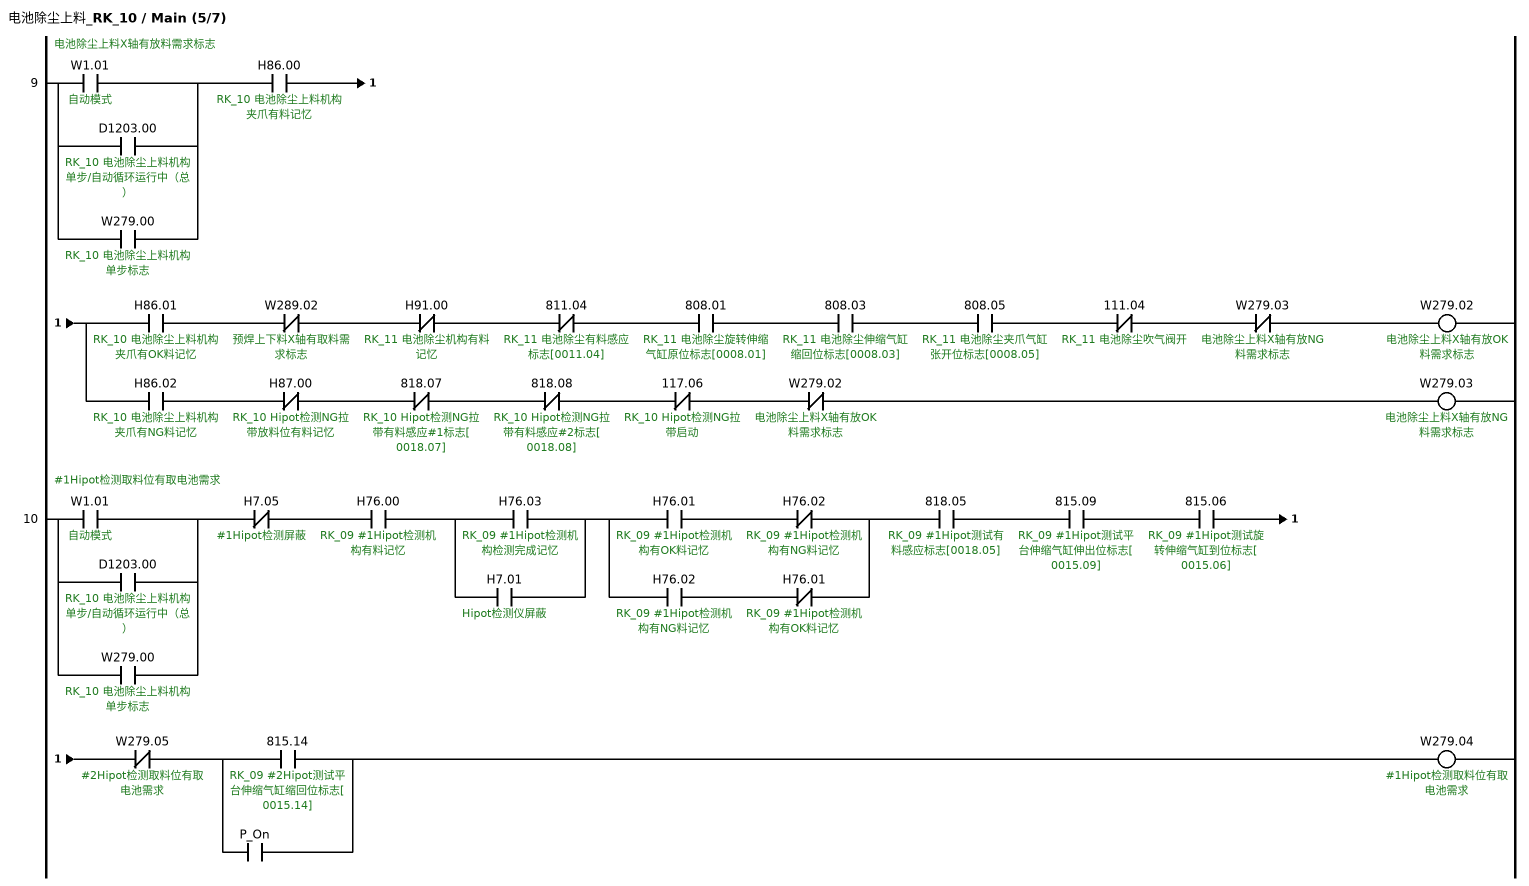
; rung 9: 电池除尘上料X轴有放料需求标志
LD W1.01  ; 自动模式
OR D1203.00  ; RK_10 电池除尘上料机构单步/自动循环运行中（总）
OR W279.00  ; RK_10 电池除尘上料机构单步标志
AND H86.00  ; RK_10 电池除尘上料机构夹爪有料记忆
OUT TR0
AND H86.01  ; RK_10 电池除尘上料机构夹爪有OK料记忆
ANDNOT W289.02  ; 预焊上下料X轴有取料需求标志
ANDNOT H91.00  ; RK_11 电池除尘机构有料记忆
ANDNOT 811.04  ; RK_11 电池除尘有料感应标志[0011.04]
AND 808.01  ; RK_11 电池除尘旋转伸缩气缸原位标志[0008.01]
AND 808.03  ; RK_11 电池除尘伸缩气缸缩回位标志[0008.03]
AND 808.05  ; RK_11 电池除尘夹爪气缸张开位标志[0008.05]
ANDNOT 111.04  ; RK_11 电池除尘吹气阀开
ANDNOT W279.03  ; 电池除尘上料X轴有放NG料需求标志
OUT W279.02  ; 电池除尘上料X轴有放OK料需求标志
LD TR0
AND H86.02  ; RK_10 电池除尘上料机构夹爪有NG料记忆
ANDNOT H87.00  ; RK_10 Hipot检测NG拉带放料位有料记忆
ANDNOT 818.07  ; RK_10 Hipot检测NG拉带有料感应#1标志[0018.07]
ANDNOT 818.08  ; RK_10 Hipot检测NG拉带有料感应#2标志[0018.08]
ANDNOT 117.06  ; RK_10 Hipot检测NG拉带启动
ANDNOT W279.02  ; 电池除尘上料X轴有放OK料需求标志
OUT W279.03  ; 电池除尘上料X轴有放NG料需求标志
; rung 10: #1Hipot检测取料位有取电池需求
LD W1.01  ; 自动模式
OR D1203.00  ; RK_10 电池除尘上料机构单步/自动循环运行中（总）
OR W279.00  ; RK_10 电池除尘上料机构单步标志
ANDNOT H7.05  ; #1Hipot检测屏蔽
AND H76.00  ; RK_09 #1Hipot检测机构有料记忆
LD H76.03  ; RK_09 #1Hipot检测机构检测完成记忆
OR H7.01  ; Hipot检测仪屏蔽
ANDLD
LD H76.01  ; RK_09 #1Hipot检测机构有OK料记忆
ANDNOT H76.02  ; RK_09 #1Hipot检测机构有NG料记忆
LD H76.02  ; RK_09 #1Hipot检测机构有NG料记忆
ANDNOT H76.01  ; RK_09 #1Hipot检测机构有OK料记忆
ORLD
ANDLD
AND 818.05  ; RK_09 #1Hipot测试有料感应标志[0018.05]
AND 815.09  ; RK_09 #1Hipot测试平台伸缩气缸伸出位标志[0015.09]
AND 815.06  ; RK_09 #1Hipot测试旋转伸缩气缸到位标志[0015.06]
ANDNOT W279.05  ; #2Hipot检测取料位有取电池需求
LD 815.14  ; RK_09 #2Hipot测试平台伸缩气缸缩回位标志[0015.14]
OR P_On
ANDLD
OUT W279.04  ; #1Hipot检测取料位有取电池需求

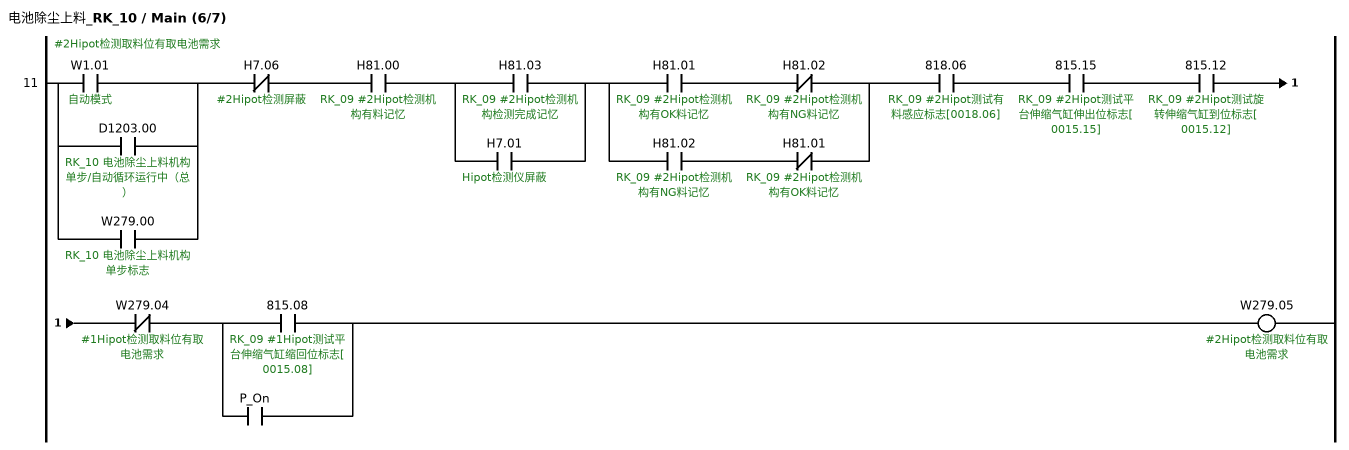
; rung 11: #2Hipot检测取料位有取电池需求
LD W1.01  ; 自动模式
OR D1203.00  ; RK_10 电池除尘上料机构单步/自动循环运行中（总）
OR W279.00  ; RK_10 电池除尘上料机构单步标志
ANDNOT H7.06  ; #2Hipot检测屏蔽
AND H81.00  ; RK_09 #2Hipot检测机构有料记忆
LD H81.03  ; RK_09 #2Hipot检测机构检测完成记忆
OR H7.01  ; Hipot检测仪屏蔽
ANDLD
LD H81.01  ; RK_09 #2Hipot检测机构有OK料记忆
ANDNOT H81.02  ; RK_09 #2Hipot检测机构有NG料记忆
LD H81.02  ; RK_09 #2Hipot检测机构有NG料记忆
ANDNOT H81.01  ; RK_09 #2Hipot检测机构有OK料记忆
ORLD
ANDLD
AND 818.06  ; RK_09 #2Hipot测试有料感应标志[0018.06]
AND 815.15  ; RK_09 #2Hipot测试平台伸缩气缸伸出位标志[0015.15]
AND 815.12  ; RK_09 #2Hipot测试旋转伸缩气缸到位标志[0015.12]
ANDNOT W279.04  ; #1Hipot检测取料位有取电池需求
LD 815.08  ; RK_09 #1Hipot测试平台伸缩气缸缩回位标志[0015.08]
OR P_On
ANDLD
OUT W279.05  ; #2Hipot检测取料位有取电池需求

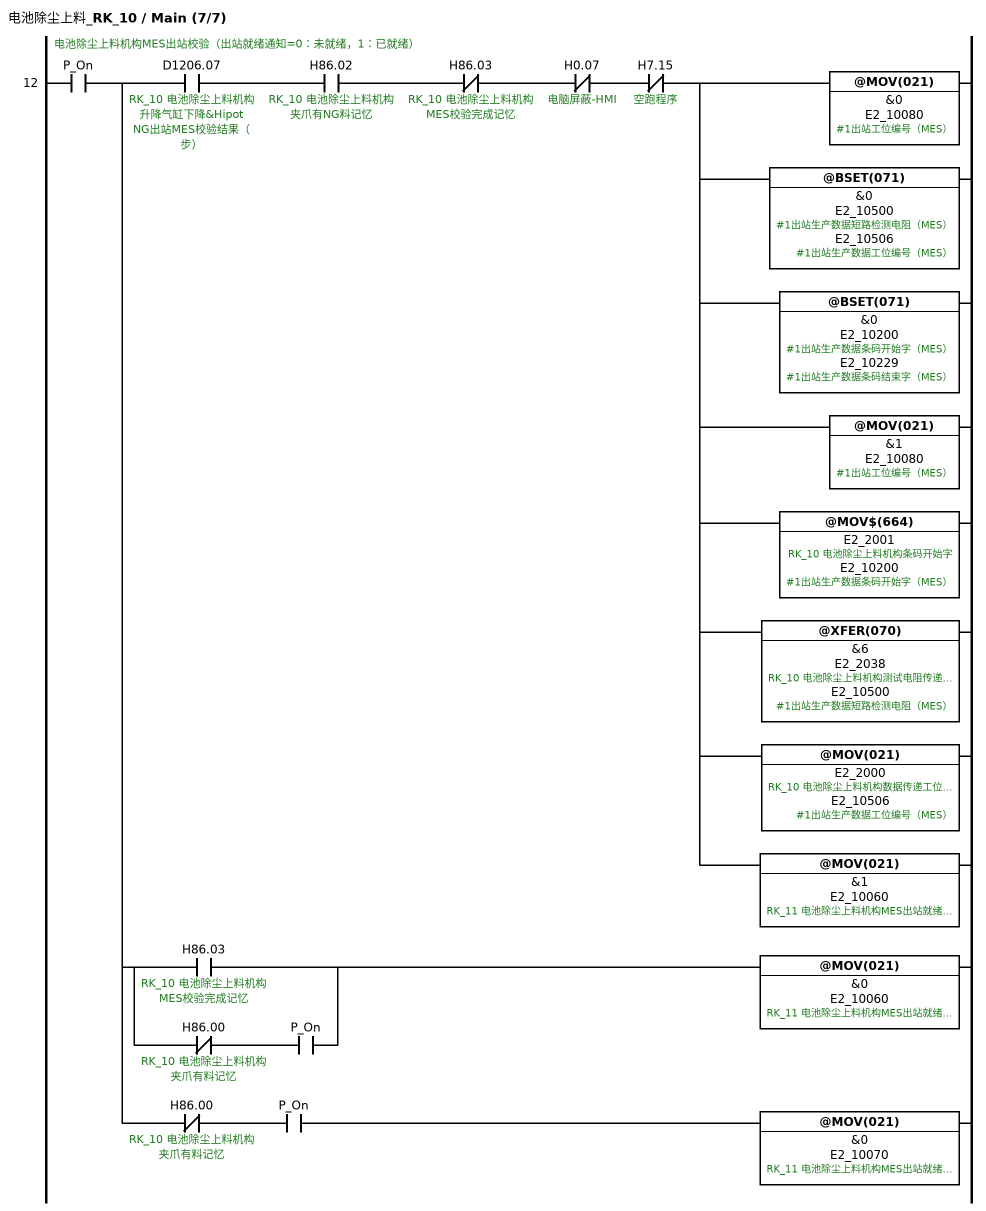
; rung 12: 电池除尘上料机构MES出站校验（出站就绪通知=0：未就绪，1：已就绪）
LD P_On
OUT TR0
AND D1206.07  ; RK_10 电池除尘上料机构升降气缸下降&Hipot NG出站MES校验结果（步）
AND H86.02  ; RK_10 电池除尘上料机构夹爪有NG料记忆
ANDNOT H86.03  ; RK_10 电池除尘上料机构MES校验完成记忆
ANDNOT H0.07  ; 电脑屏蔽-HMI
ANDNOT H7.15  ; 空跑程序
@MOV(021) &0 E2_10080  ; #1出站工位编号（MES）
@BSET(071) &0 E2_10500 E2_10506  ; #1出站生产数据短路检测电阻（MES）, #1出站生产数据工位编号（MES）
@BSET(071) &0 E2_10200 E2_10229  ; #1出站生产数据条码开始字（MES）, #1出站生产数据条码结束字（MES）
@MOV(021) &1 E2_10080  ; #1出站工位编号（MES）
@MOV$(664) E2_2001 E2_10200  ; RK_10 电池除尘上料机构条码开始字, #1出站生产数据条码开始字（MES）
@XFER(070) &6 E2_2038 E2_10500  ; RK_10 电池除尘上料机构测试电阻传递（Float）, #1出站生产数据短路检测电阻（MES）
@MOV(021) E2_2000 E2_10506  ; RK_10 电池除尘上料机构数据传递工位编号, #1出站生产数据工位编号（MES）
@MOV(021) &1 E2_10060  ; RK_11 电池除尘上料机构MES出站就绪通知
LD TR0
LD H86.03  ; RK_10 电池除尘上料机构MES校验完成记忆
LDNOT H86.00  ; RK_10 电池除尘上料机构夹爪有料记忆
AND P_On
ORLD
ANDLD
@MOV(021) &0 E2_10060  ; RK_11 电池除尘上料机构MES出站就绪通知
LD TR0
ANDNOT H86.00  ; RK_10 电池除尘上料机构夹爪有料记忆
AND P_On
@MOV(021) &0 E2_10070  ; RK_11 电池除尘上料机构MES出站就绪确认

### Section 手动

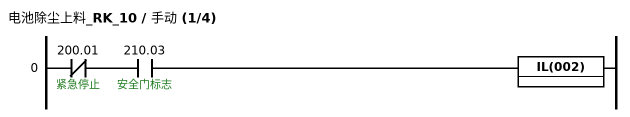
; rung 0
LDNOT 200.01  ; 紧急停止
AND 210.03  ; 安全门标志
IL(002)

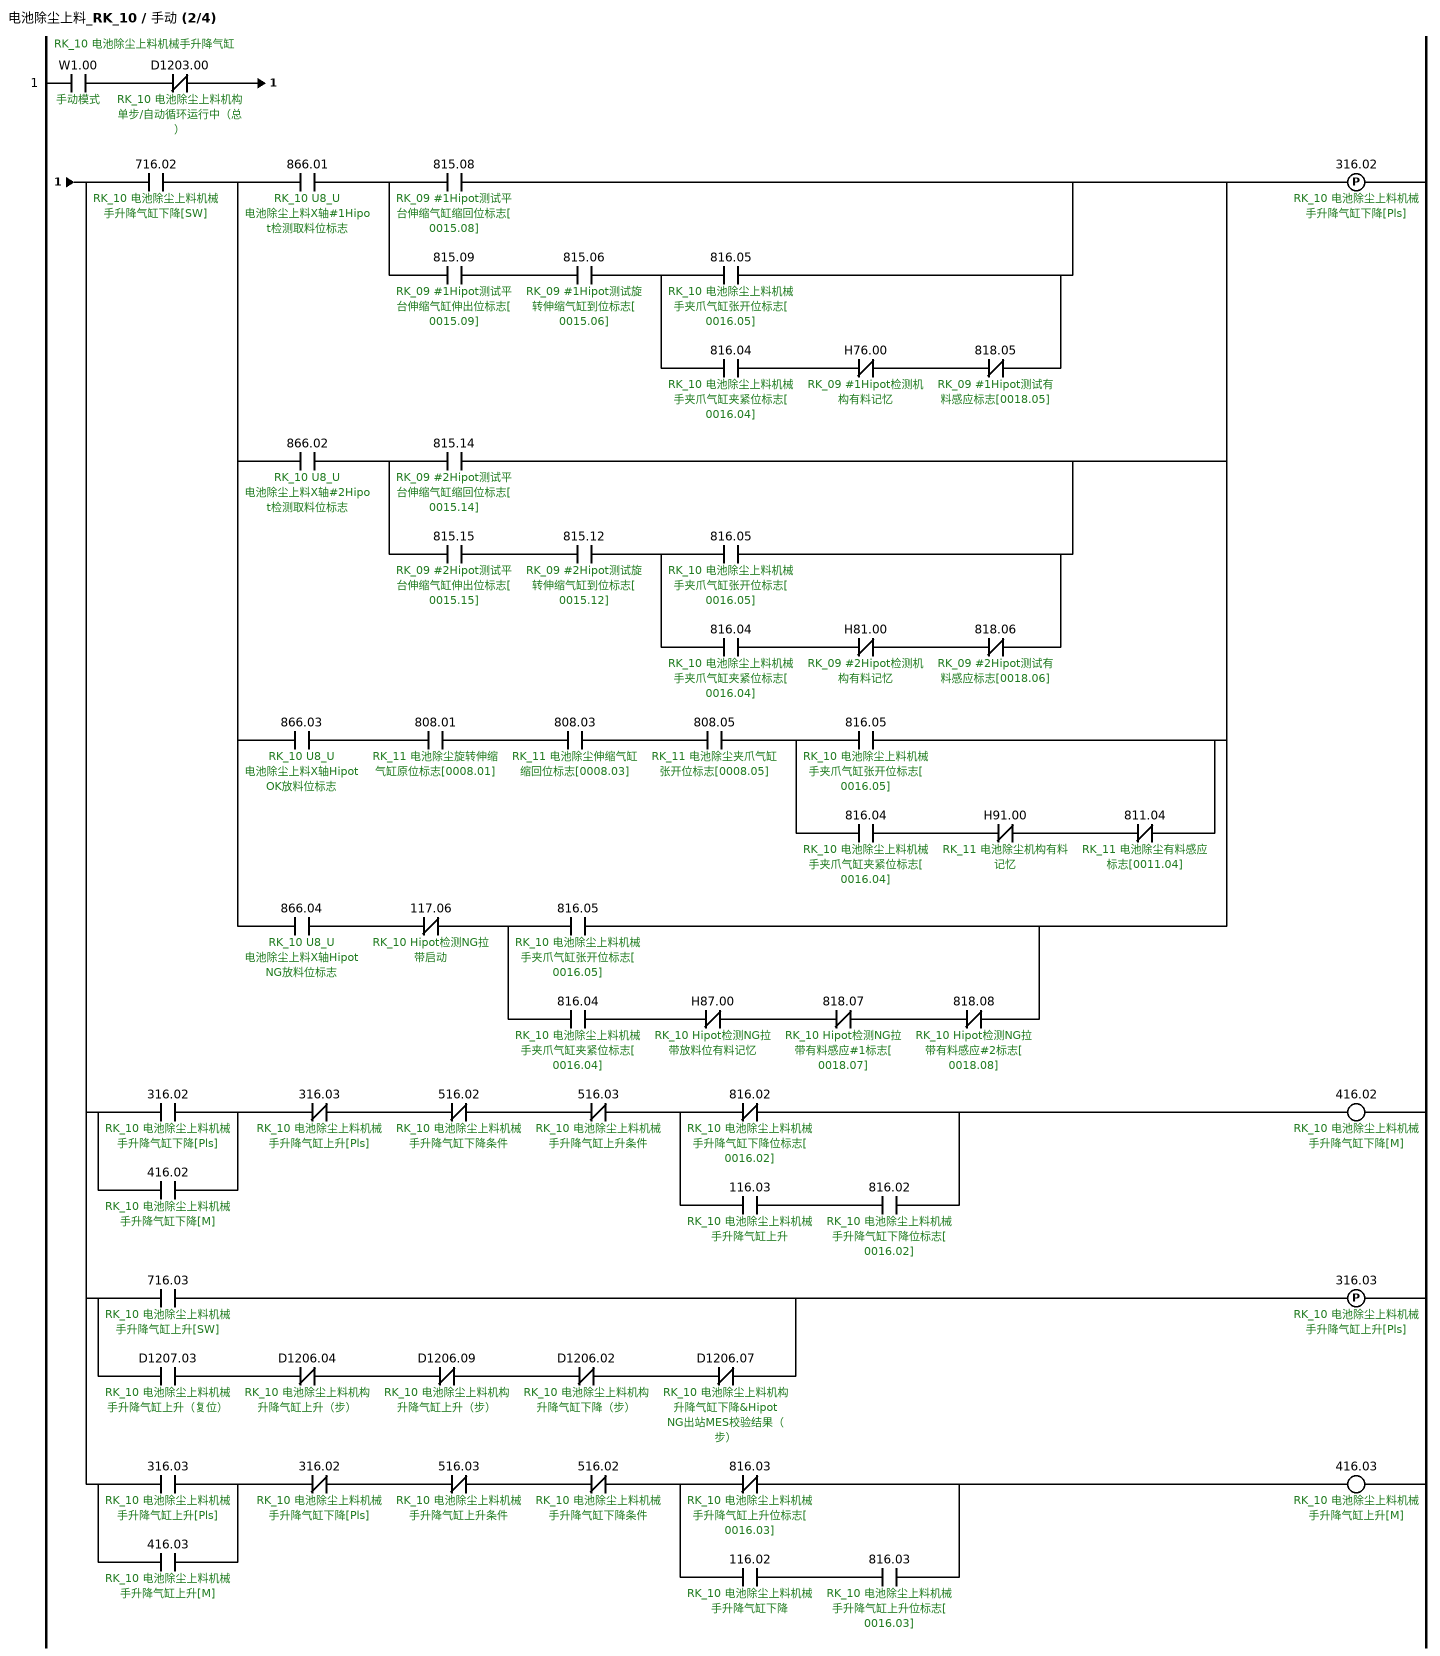
; rung 1: RK_10 电池除尘上料机械手升降气缸
LD W1.00  ; 手动模式
ANDNOT D1203.00  ; RK_10 电池除尘上料机构单步/自动循环运行中（总）
OUT TR0
AND 716.02  ; RK_10 电池除尘上料机械手升降气缸下降[SW]
LD 866.01  ; RK_10 U8_U 电池除尘上料X轴#1Hipot检测取料位标志
LD 815.08  ; RK_09 #1Hipot测试平台伸缩气缸缩回位标志[0015.08]
LD 815.09  ; RK_09 #1Hipot测试平台伸缩气缸伸出位标志[0015.09]
AND 815.06  ; RK_09 #1Hipot测试旋转伸缩气缸到位标志[0015.06]
LD 816.05  ; RK_10 电池除尘上料机械手夹爪气缸张开位标志[0016.05]
LD 816.04  ; RK_10 电池除尘上料机械手夹爪气缸夹紧位标志[0016.04]
ANDNOT H76.00  ; RK_09 #1Hipot检测机构有料记忆
ANDNOT 818.05  ; RK_09 #1Hipot测试有料感应标志[0018.05]
ORLD
ANDLD
ORLD
ANDLD
LD 866.02  ; RK_10 U8_U 电池除尘上料X轴#2Hipot检测取料位标志
LD 815.14  ; RK_09 #2Hipot测试平台伸缩气缸缩回位标志[0015.14]
LD 815.15  ; RK_09 #2Hipot测试平台伸缩气缸伸出位标志[0015.15]
AND 815.12  ; RK_09 #2Hipot测试旋转伸缩气缸到位标志[0015.12]
LD 816.05  ; RK_10 电池除尘上料机械手夹爪气缸张开位标志[0016.05]
LD 816.04  ; RK_10 电池除尘上料机械手夹爪气缸夹紧位标志[0016.04]
ANDNOT H81.00  ; RK_09 #2Hipot检测机构有料记忆
ANDNOT 818.06  ; RK_09 #2Hipot测试有料感应标志[0018.06]
ORLD
ANDLD
ORLD
ANDLD
ORLD
LD 866.03  ; RK_10 U8_U 电池除尘上料X轴Hipot OK放料位标志
AND 808.01  ; RK_11 电池除尘旋转伸缩气缸原位标志[0008.01]
AND 808.03  ; RK_11 电池除尘伸缩气缸缩回位标志[0008.03]
AND 808.05  ; RK_11 电池除尘夹爪气缸张开位标志[0008.05]
LD 816.05  ; RK_10 电池除尘上料机械手夹爪气缸张开位标志[0016.05]
LD 816.04  ; RK_10 电池除尘上料机械手夹爪气缸夹紧位标志[0016.04]
ANDNOT H91.00  ; RK_11 电池除尘机构有料记忆
ANDNOT 811.04  ; RK_11 电池除尘有料感应标志[0011.04]
ORLD
ANDLD
ORLD
LD 866.04  ; RK_10 U8_U 电池除尘上料X轴Hipot NG放料位标志
ANDNOT 117.06  ; RK_10 Hipot检测NG拉带启动
LD 816.05  ; RK_10 电池除尘上料机械手夹爪气缸张开位标志[0016.05]
LD 816.04  ; RK_10 电池除尘上料机械手夹爪气缸夹紧位标志[0016.04]
ANDNOT H87.00  ; RK_10 Hipot检测NG拉带放料位有料记忆
ANDNOT 818.07  ; RK_10 Hipot检测NG拉带有料感应#1标志[0018.07]
ANDNOT 818.08  ; RK_10 Hipot检测NG拉带有料感应#2标志[0018.08]
ORLD
ANDLD
ORLD
ANDLD
DIFU(013) 316.02  ; RK_10 电池除尘上料机械手升降气缸下降[Pls]
LD TR0
LD 316.02  ; RK_10 电池除尘上料机械手升降气缸下降[Pls]
OR 416.02  ; RK_10 电池除尘上料机械手升降气缸下降[M]
ANDLD
ANDNOT 316.03  ; RK_10 电池除尘上料机械手升降气缸上升[Pls]
ANDNOT 516.02  ; RK_10 电池除尘上料机械手升降气缸下降条件
ANDNOT 516.03  ; RK_10 电池除尘上料机械手升降气缸上升条件
LDNOT 816.02  ; RK_10 电池除尘上料机械手升降气缸下降位标志[0016.02]
LD 116.03  ; RK_10 电池除尘上料机械手升降气缸上升
AND 816.02  ; RK_10 电池除尘上料机械手升降气缸下降位标志[0016.02]
ORLD
ANDLD
OUT 416.02  ; RK_10 电池除尘上料机械手升降气缸下降[M]
LD TR0
LD 716.03  ; RK_10 电池除尘上料机械手升降气缸上升[SW]
LD D1207.03  ; RK_10 电池除尘上料机械手升降气缸上升（复位）
ANDNOT D1206.04  ; RK_10 电池除尘上料机构升降气缸上升（步）
ANDNOT D1206.09  ; RK_10 电池除尘上料机构升降气缸上升（步）
ANDNOT D1206.02  ; RK_10 电池除尘上料机构升降气缸下降（步）
ANDNOT D1206.07  ; RK_10 电池除尘上料机构升降气缸下降&Hipot NG出站MES校验结果（步）
ORLD
ANDLD
DIFU(013) 316.03  ; RK_10 电池除尘上料机械手升降气缸上升[Pls]
LD TR0
LD 316.03  ; RK_10 电池除尘上料机械手升降气缸上升[Pls]
OR 416.03  ; RK_10 电池除尘上料机械手升降气缸上升[M]
ANDLD
ANDNOT 316.02  ; RK_10 电池除尘上料机械手升降气缸下降[Pls]
ANDNOT 516.03  ; RK_10 电池除尘上料机械手升降气缸上升条件
ANDNOT 516.02  ; RK_10 电池除尘上料机械手升降气缸下降条件
LDNOT 816.03  ; RK_10 电池除尘上料机械手升降气缸上升位标志[0016.03]
LD 116.02  ; RK_10 电池除尘上料机械手升降气缸下降
AND 816.03  ; RK_10 电池除尘上料机械手升降气缸上升位标志[0016.03]
ORLD
ANDLD
OUT 416.03  ; RK_10 电池除尘上料机械手升降气缸上升[M]

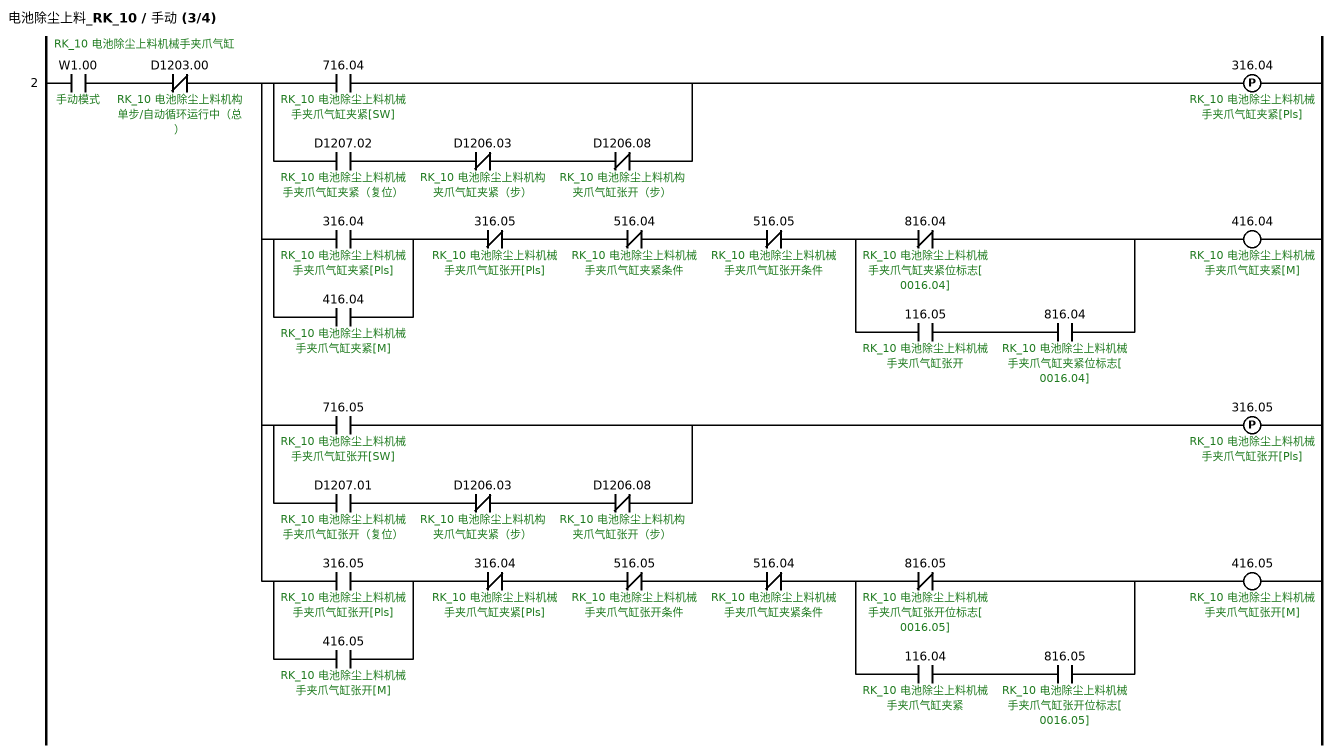
; rung 2: RK_10 电池除尘上料机械手夹爪气缸
LD W1.00  ; 手动模式
ANDNOT D1203.00  ; RK_10 电池除尘上料机构单步/自动循环运行中（总）
OUT TR0
LD 716.04  ; RK_10 电池除尘上料机械手夹爪气缸夹紧[SW]
LD D1207.02  ; RK_10 电池除尘上料机械手夹爪气缸夹紧（复位）
ANDNOT D1206.03  ; RK_10 电池除尘上料机构夹爪气缸夹紧（步）
ANDNOT D1206.08  ; RK_10 电池除尘上料机构夹爪气缸张开（步）
ORLD
ANDLD
DIFU(013) 316.04  ; RK_10 电池除尘上料机械手夹爪气缸夹紧[Pls]
LD TR0
LD 316.04  ; RK_10 电池除尘上料机械手夹爪气缸夹紧[Pls]
OR 416.04  ; RK_10 电池除尘上料机械手夹爪气缸夹紧[M]
ANDLD
ANDNOT 316.05  ; RK_10 电池除尘上料机械手夹爪气缸张开[Pls]
ANDNOT 516.04  ; RK_10 电池除尘上料机械手夹爪气缸夹紧条件
ANDNOT 516.05  ; RK_10 电池除尘上料机械手夹爪气缸张开条件
LDNOT 816.04  ; RK_10 电池除尘上料机械手夹爪气缸夹紧位标志[0016.04]
LD 116.05  ; RK_10 电池除尘上料机械手夹爪气缸张开
AND 816.04  ; RK_10 电池除尘上料机械手夹爪气缸夹紧位标志[0016.04]
ORLD
ANDLD
OUT 416.04  ; RK_10 电池除尘上料机械手夹爪气缸夹紧[M]
LD TR0
LD 716.05  ; RK_10 电池除尘上料机械手夹爪气缸张开[SW]
LD D1207.01  ; RK_10 电池除尘上料机械手夹爪气缸张开（复位）
ANDNOT D1206.03  ; RK_10 电池除尘上料机构夹爪气缸夹紧（步）
ANDNOT D1206.08  ; RK_10 电池除尘上料机构夹爪气缸张开（步）
ORLD
ANDLD
DIFU(013) 316.05  ; RK_10 电池除尘上料机械手夹爪气缸张开[Pls]
LD TR0
LD 316.05  ; RK_10 电池除尘上料机械手夹爪气缸张开[Pls]
OR 416.05  ; RK_10 电池除尘上料机械手夹爪气缸张开[M]
ANDLD
ANDNOT 316.04  ; RK_10 电池除尘上料机械手夹爪气缸夹紧[Pls]
ANDNOT 516.05  ; RK_10 电池除尘上料机械手夹爪气缸张开条件
ANDNOT 516.04  ; RK_10 电池除尘上料机械手夹爪气缸夹紧条件
LDNOT 816.05  ; RK_10 电池除尘上料机械手夹爪气缸张开位标志[0016.05]
LD 116.04  ; RK_10 电池除尘上料机械手夹爪气缸夹紧
AND 816.05  ; RK_10 电池除尘上料机械手夹爪气缸张开位标志[0016.05]
ORLD
ANDLD
OUT 416.05  ; RK_10 电池除尘上料机械手夹爪气缸张开[M]

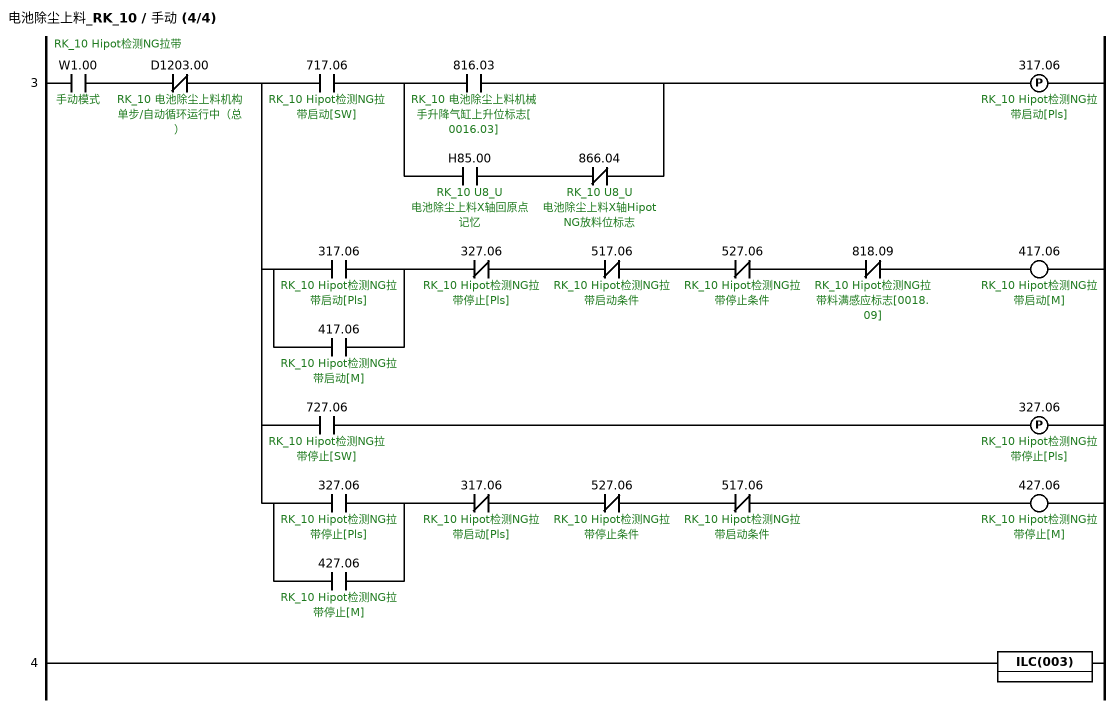
; rung 3: RK_10 Hipot检测NG拉带
LD W1.00  ; 手动模式
ANDNOT D1203.00  ; RK_10 电池除尘上料机构单步/自动循环运行中（总）
OUT TR0
AND 717.06  ; RK_10 Hipot检测NG拉带启动[SW]
LD 816.03  ; RK_10 电池除尘上料机械手升降气缸上升位标志[0016.03]
LD H85.00  ; RK_10 U8_U 电池除尘上料X轴回原点记忆
ANDNOT 866.04  ; RK_10 U8_U 电池除尘上料X轴Hipot NG放料位标志
ORLD
ANDLD
DIFU(013) 317.06  ; RK_10 Hipot检测NG拉带启动[Pls]
LD TR0
LD 317.06  ; RK_10 Hipot检测NG拉带启动[Pls]
OR 417.06  ; RK_10 Hipot检测NG拉带启动[M]
ANDLD
ANDNOT 327.06  ; RK_10 Hipot检测NG拉带停止[Pls]
ANDNOT 517.06  ; RK_10 Hipot检测NG拉带启动条件
ANDNOT 527.06  ; RK_10 Hipot检测NG拉带停止条件
ANDNOT 818.09  ; RK_10 Hipot检测NG拉带料满感应标志[0018.09]
OUT 417.06  ; RK_10 Hipot检测NG拉带启动[M]
LD TR0
AND 727.06  ; RK_10 Hipot检测NG拉带停止[SW]
DIFU(013) 327.06  ; RK_10 Hipot检测NG拉带停止[Pls]
LD TR0
LD 327.06  ; RK_10 Hipot检测NG拉带停止[Pls]
OR 427.06  ; RK_10 Hipot检测NG拉带停止[M]
ANDLD
ANDNOT 317.06  ; RK_10 Hipot检测NG拉带启动[Pls]
ANDNOT 527.06  ; RK_10 Hipot检测NG拉带停止条件
ANDNOT 517.06  ; RK_10 Hipot检测NG拉带启动条件
OUT 427.06  ; RK_10 Hipot检测NG拉带停止[M]
; rung 4
ILC(003)

### Section 自动

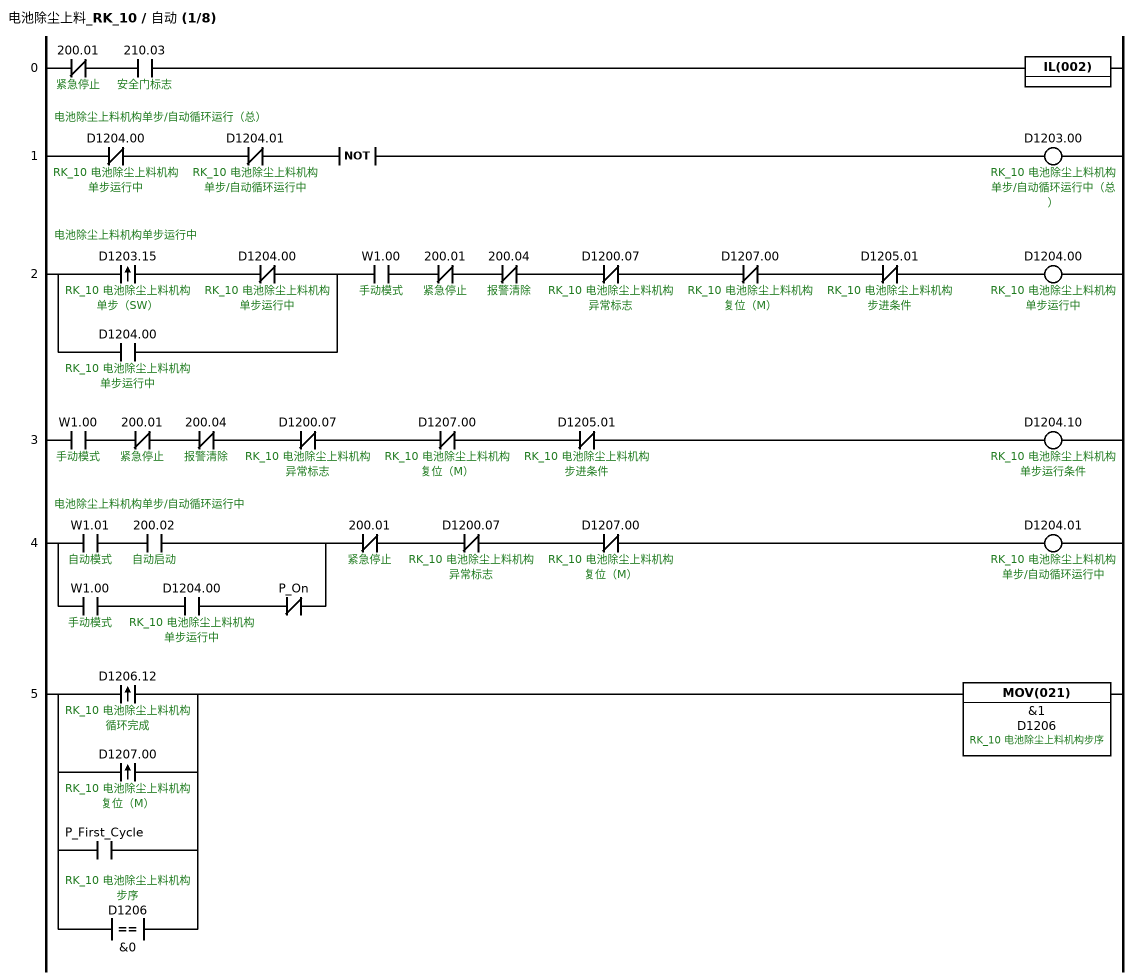
; rung 0
LDNOT 200.01  ; 紧急停止
AND 210.03  ; 安全门标志
IL(002)
; rung 1: 电池除尘上料机构单步/自动循环运行（总）
LDNOT D1204.00  ; RK_10 电池除尘上料机构单步运行中
ANDNOT D1204.01  ; RK_10 电池除尘上料机构单步/自动循环运行中
NOT(520)
OUT D1203.00  ; RK_10 电池除尘上料机构单步/自动循环运行中（总）
; rung 2: 电池除尘上料机构单步运行中
@LD D1203.15  ; RK_10 电池除尘上料机构单步（SW）
ANDNOT D1204.00  ; RK_10 电池除尘上料机构单步运行中
OR D1204.00  ; RK_10 电池除尘上料机构单步运行中
AND W1.00  ; 手动模式
ANDNOT 200.01  ; 紧急停止
ANDNOT 200.04  ; 报警清除
ANDNOT D1200.07  ; RK_10 电池除尘上料机构异常标志
ANDNOT D1207.00  ; RK_10 电池除尘上料机构复位（M）
ANDNOT D1205.01  ; RK_10 电池除尘上料机构步进条件
OUT D1204.00  ; RK_10 电池除尘上料机构单步运行中
; rung 3
LD W1.00  ; 手动模式
ANDNOT 200.01  ; 紧急停止
ANDNOT 200.04  ; 报警清除
ANDNOT D1200.07  ; RK_10 电池除尘上料机构异常标志
ANDNOT D1207.00  ; RK_10 电池除尘上料机构复位（M）
ANDNOT D1205.01  ; RK_10 电池除尘上料机构步进条件
OUT D1204.10  ; RK_10 电池除尘上料机构单步运行条件
; rung 4: 电池除尘上料机构单步/自动循环运行中
LD W1.01  ; 自动模式
AND 200.02  ; 自动启动
LD W1.00  ; 手动模式
AND D1204.00  ; RK_10 电池除尘上料机构单步运行中
ANDNOT P_On
ORLD
ANDNOT 200.01  ; 紧急停止
ANDNOT D1200.07  ; RK_10 电池除尘上料机构异常标志
ANDNOT D1207.00  ; RK_10 电池除尘上料机构复位（M）
OUT D1204.01  ; RK_10 电池除尘上料机构单步/自动循环运行中
; rung 5
@LD D1206.12  ; RK_10 电池除尘上料机构循环完成
@OR D1207.00  ; RK_10 电池除尘上料机构复位（M）
OR P_First_Cycle
OR=(300) D1206 &0  ; RK_10 电池除尘上料机构步序
MOV(021) &1 D1206  ; RK_10 电池除尘上料机构步序

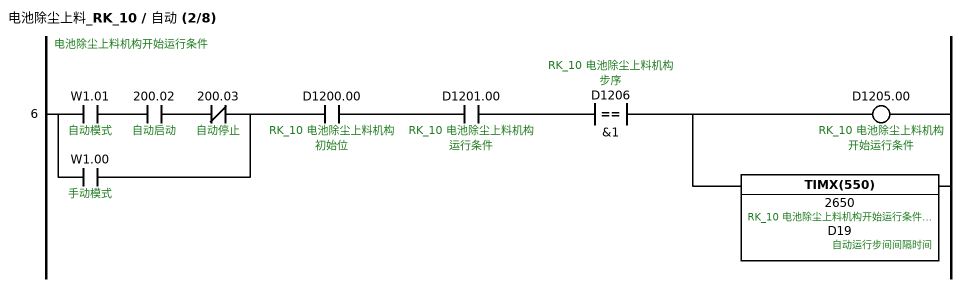
; rung 6: 电池除尘上料机构开始运行条件
LD W1.01  ; 自动模式
AND 200.02  ; 自动启动
ANDNOT 200.03  ; 自动停止
OR W1.00  ; 手动模式
AND D1200.00  ; RK_10 电池除尘上料机构初始位
AND D1201.00  ; RK_10 电池除尘上料机构运行条件
AND=(300) D1206 &1  ; RK_10 电池除尘上料机构步序
OUT D1205.00  ; RK_10 电池除尘上料机构开始运行条件
TIMX(550) 2650 D19  ; 自动运行步间间隔时间, RK_10 电池除尘上料机构开始运行条件延时

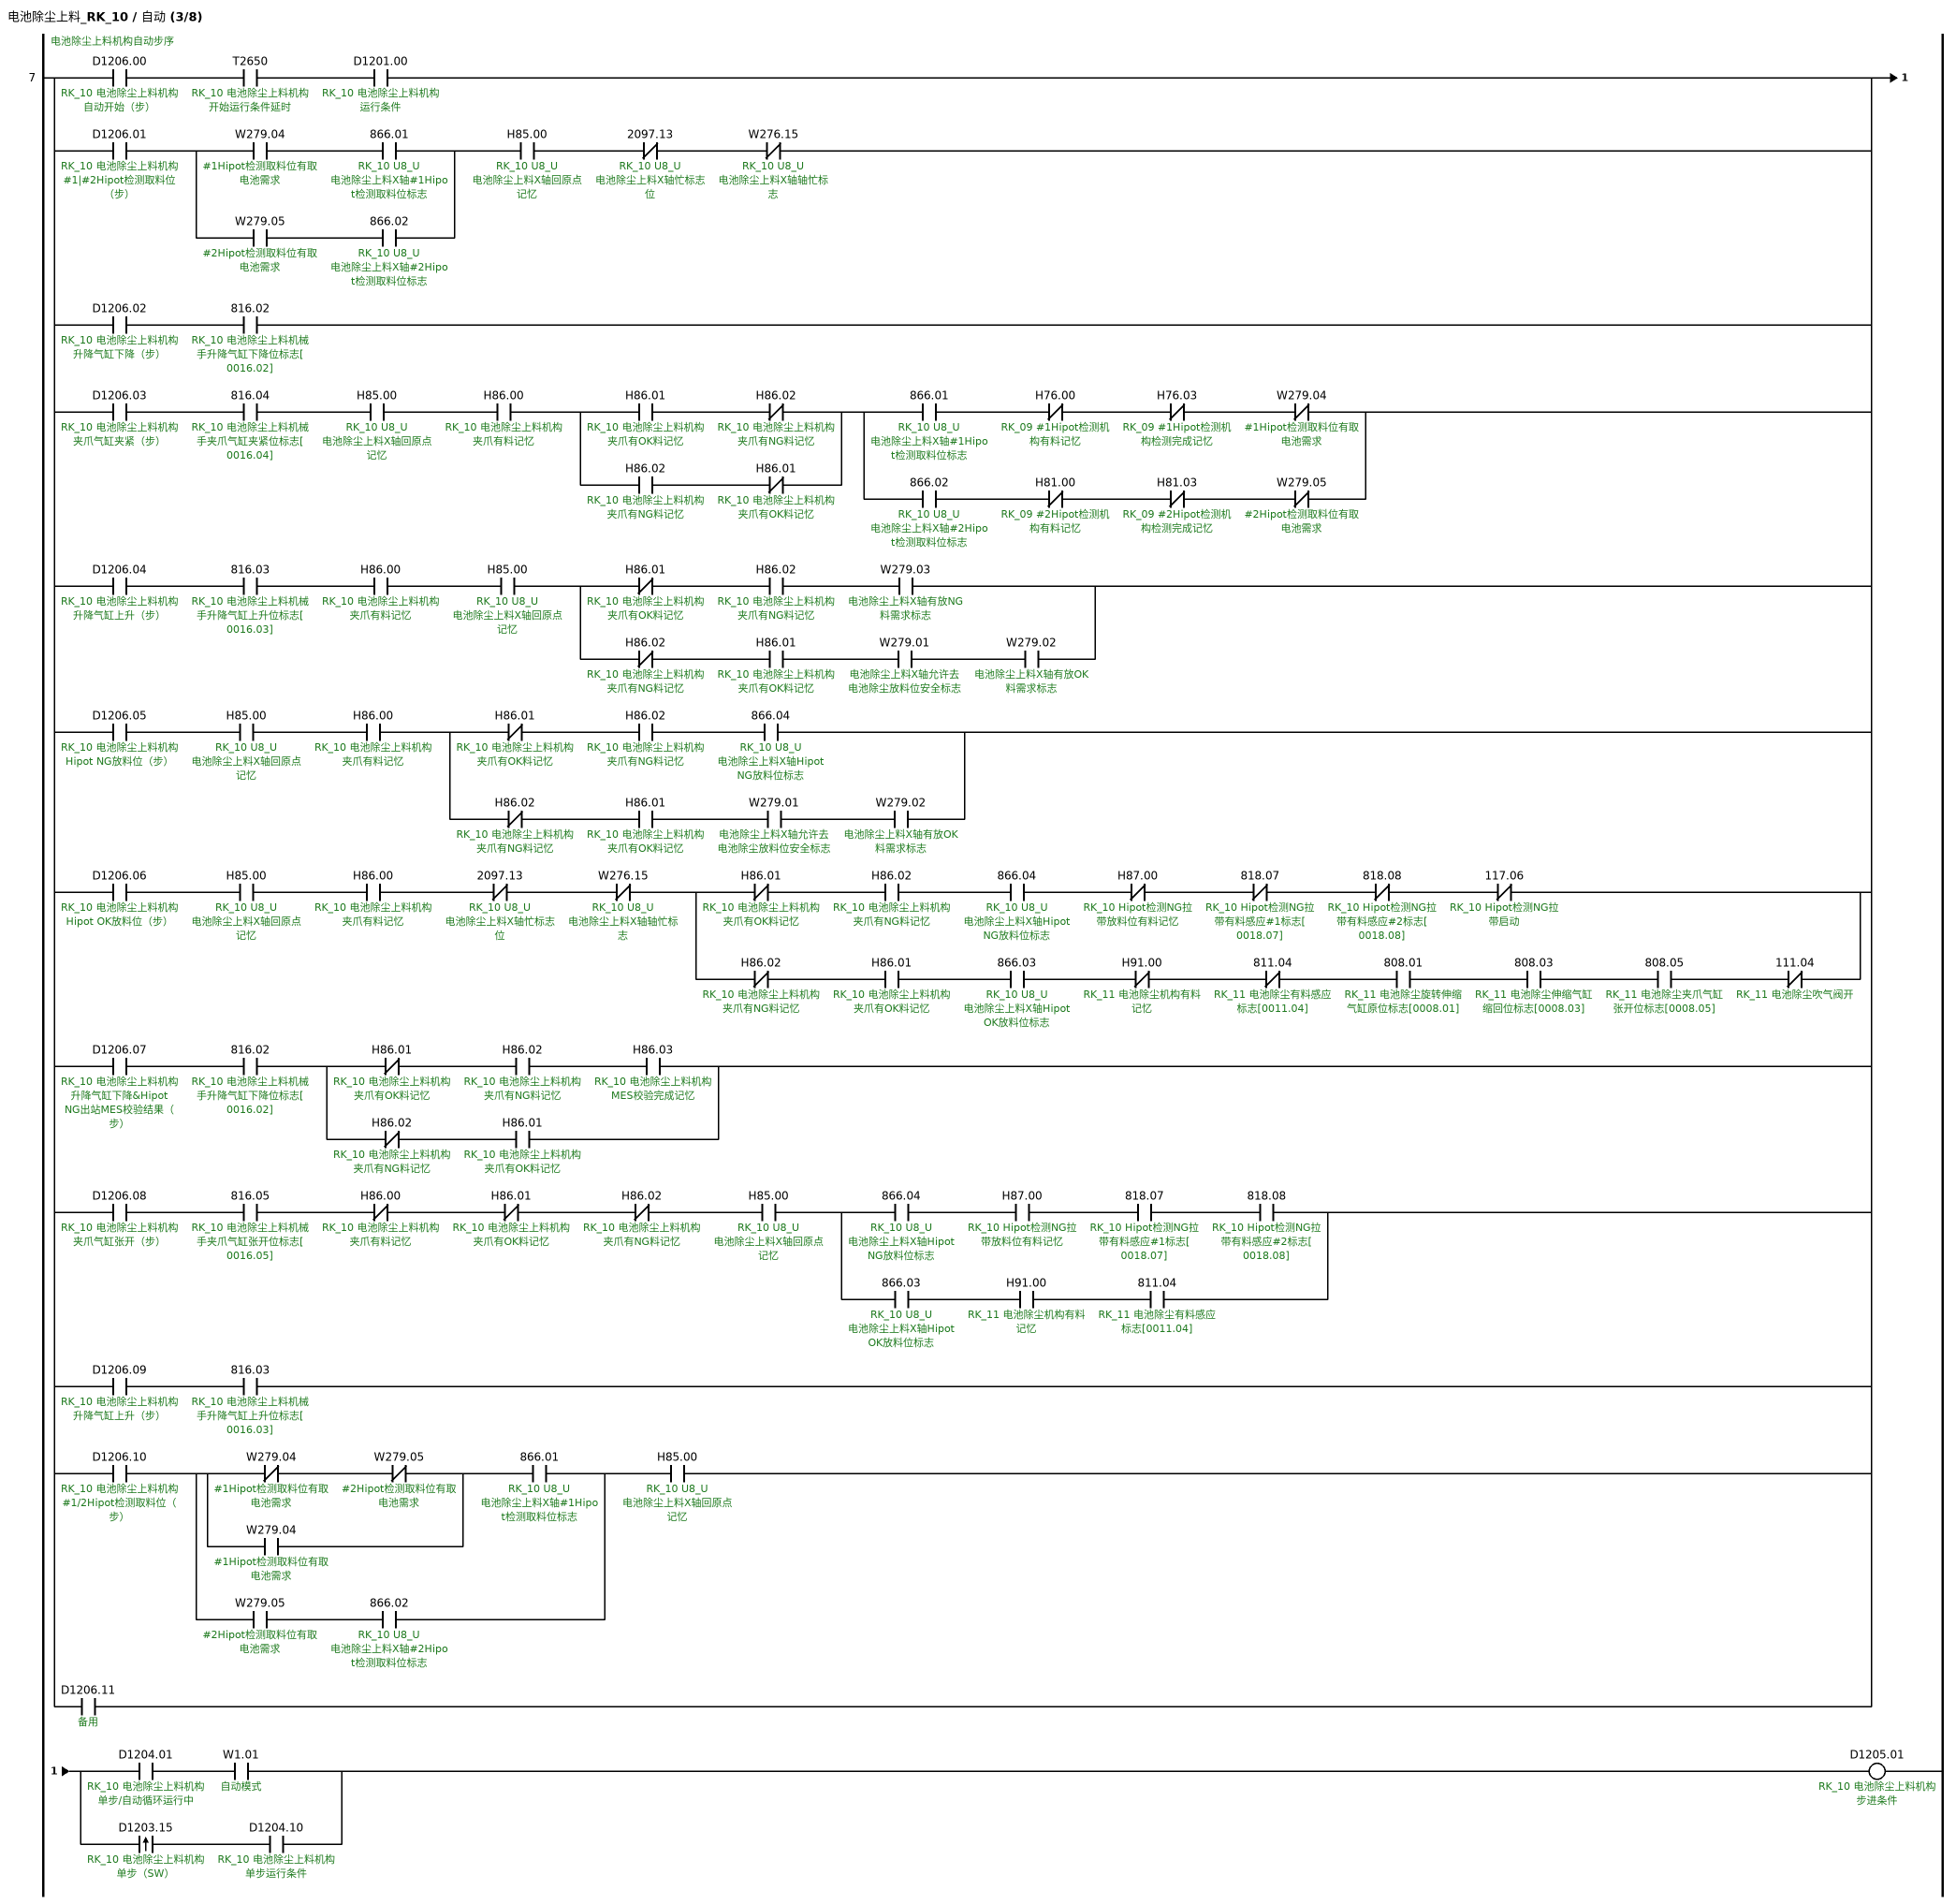
; rung 7: 电池除尘上料机构自动步序
LD D1206.00  ; RK_10 电池除尘上料机构自动开始（步）
AND T2650  ; RK_10 电池除尘上料机构开始运行条件延时
AND D1201.00  ; RK_10 电池除尘上料机构运行条件
LD D1206.01  ; RK_10 电池除尘上料机构#1|#2Hipot检测取料位（步）
LD W279.04  ; #1Hipot检测取料位有取电池需求
AND 866.01  ; RK_10 U8_U 电池除尘上料X轴#1Hipot检测取料位标志
LD W279.05  ; #2Hipot检测取料位有取电池需求
AND 866.02  ; RK_10 U8_U 电池除尘上料X轴#2Hipot检测取料位标志
ORLD
ANDLD
AND H85.00  ; RK_10 U8_U 电池除尘上料X轴回原点记忆
ANDNOT 2097.13  ; RK_10 U8_U 电池除尘上料X轴忙标志位
ANDNOT W276.15  ; RK_10 U8_U 电池除尘上料X轴轴忙标志
ORLD
LD D1206.02  ; RK_10 电池除尘上料机构升降气缸下降（步）
AND 816.02  ; RK_10 电池除尘上料机械手升降气缸下降位标志[0016.02]
ORLD
LD D1206.03  ; RK_10 电池除尘上料机构夹爪气缸夹紧（步）
AND 816.04  ; RK_10 电池除尘上料机械手夹爪气缸夹紧位标志[0016.04]
AND H85.00  ; RK_10 U8_U 电池除尘上料X轴回原点记忆
AND H86.00  ; RK_10 电池除尘上料机构夹爪有料记忆
LD H86.01  ; RK_10 电池除尘上料机构夹爪有OK料记忆
ANDNOT H86.02  ; RK_10 电池除尘上料机构夹爪有NG料记忆
LD H86.02  ; RK_10 电池除尘上料机构夹爪有NG料记忆
ANDNOT H86.01  ; RK_10 电池除尘上料机构夹爪有OK料记忆
ORLD
ANDLD
LD 866.01  ; RK_10 U8_U 电池除尘上料X轴#1Hipot检测取料位标志
ANDNOT H76.00  ; RK_09 #1Hipot检测机构有料记忆
ANDNOT H76.03  ; RK_09 #1Hipot检测机构检测完成记忆
ANDNOT W279.04  ; #1Hipot检测取料位有取电池需求
LD 866.02  ; RK_10 U8_U 电池除尘上料X轴#2Hipot检测取料位标志
ANDNOT H81.00  ; RK_09 #2Hipot检测机构有料记忆
ANDNOT H81.03  ; RK_09 #2Hipot检测机构检测完成记忆
ANDNOT W279.05  ; #2Hipot检测取料位有取电池需求
ORLD
ANDLD
ORLD
LD D1206.04  ; RK_10 电池除尘上料机构升降气缸上升（步）
AND 816.03  ; RK_10 电池除尘上料机械手升降气缸上升位标志[0016.03]
AND H86.00  ; RK_10 电池除尘上料机构夹爪有料记忆
AND H85.00  ; RK_10 U8_U 电池除尘上料X轴回原点记忆
LDNOT H86.01  ; RK_10 电池除尘上料机构夹爪有OK料记忆
AND H86.02  ; RK_10 电池除尘上料机构夹爪有NG料记忆
AND W279.03  ; 电池除尘上料X轴有放NG料需求标志
LDNOT H86.02  ; RK_10 电池除尘上料机构夹爪有NG料记忆
AND H86.01  ; RK_10 电池除尘上料机构夹爪有OK料记忆
AND W279.01  ; 电池除尘上料X轴允许去电池除尘放料位安全标志
AND W279.02  ; 电池除尘上料X轴有放OK料需求标志
ORLD
ANDLD
ORLD
LD D1206.05  ; RK_10 电池除尘上料机构Hipot NG放料位（步）
AND H85.00  ; RK_10 U8_U 电池除尘上料X轴回原点记忆
AND H86.00  ; RK_10 电池除尘上料机构夹爪有料记忆
LDNOT H86.01  ; RK_10 电池除尘上料机构夹爪有OK料记忆
AND H86.02  ; RK_10 电池除尘上料机构夹爪有NG料记忆
AND 866.04  ; RK_10 U8_U 电池除尘上料X轴Hipot NG放料位标志
LDNOT H86.02  ; RK_10 电池除尘上料机构夹爪有NG料记忆
AND H86.01  ; RK_10 电池除尘上料机构夹爪有OK料记忆
AND W279.01  ; 电池除尘上料X轴允许去电池除尘放料位安全标志
AND W279.02  ; 电池除尘上料X轴有放OK料需求标志
ORLD
ANDLD
ORLD
LD D1206.06  ; RK_10 电池除尘上料机构Hipot OK放料位（步）
AND H85.00  ; RK_10 U8_U 电池除尘上料X轴回原点记忆
AND H86.00  ; RK_10 电池除尘上料机构夹爪有料记忆
ANDNOT 2097.13  ; RK_10 U8_U 电池除尘上料X轴忙标志位
ANDNOT W276.15  ; RK_10 U8_U 电池除尘上料X轴轴忙标志
LDNOT H86.01  ; RK_10 电池除尘上料机构夹爪有OK料记忆
AND H86.02  ; RK_10 电池除尘上料机构夹爪有NG料记忆
AND 866.04  ; RK_10 U8_U 电池除尘上料X轴Hipot NG放料位标志
ANDNOT H87.00  ; RK_10 Hipot检测NG拉带放料位有料记忆
ANDNOT 818.07  ; RK_10 Hipot检测NG拉带有料感应#1标志[0018.07]
ANDNOT 818.08  ; RK_10 Hipot检测NG拉带有料感应#2标志[0018.08]
ANDNOT 117.06  ; RK_10 Hipot检测NG拉带启动
LDNOT H86.02  ; RK_10 电池除尘上料机构夹爪有NG料记忆
AND H86.01  ; RK_10 电池除尘上料机构夹爪有OK料记忆
AND 866.03  ; RK_10 U8_U 电池除尘上料X轴Hipot OK放料位标志
ANDNOT H91.00  ; RK_11 电池除尘机构有料记忆
ANDNOT 811.04  ; RK_11 电池除尘有料感应标志[0011.04]
AND 808.01  ; RK_11 电池除尘旋转伸缩气缸原位标志[0008.01]
AND 808.03  ; RK_11 电池除尘伸缩气缸缩回位标志[0008.03]
AND 808.05  ; RK_11 电池除尘夹爪气缸张开位标志[0008.05]
ANDNOT 111.04  ; RK_11 电池除尘吹气阀开
ORLD
ANDLD
ORLD
LD D1206.07  ; RK_10 电池除尘上料机构升降气缸下降&Hipot NG出站MES校验结果（步）
AND 816.02  ; RK_10 电池除尘上料机械手升降气缸下降位标志[0016.02]
LDNOT H86.01  ; RK_10 电池除尘上料机构夹爪有OK料记忆
AND H86.02  ; RK_10 电池除尘上料机构夹爪有NG料记忆
AND H86.03  ; RK_10 电池除尘上料机构MES校验完成记忆
LDNOT H86.02  ; RK_10 电池除尘上料机构夹爪有NG料记忆
AND H86.01  ; RK_10 电池除尘上料机构夹爪有OK料记忆
ORLD
ANDLD
ORLD
LD D1206.08  ; RK_10 电池除尘上料机构夹爪气缸张开（步）
AND 816.05  ; RK_10 电池除尘上料机械手夹爪气缸张开位标志[0016.05]
ANDNOT H86.00  ; RK_10 电池除尘上料机构夹爪有料记忆
ANDNOT H86.01  ; RK_10 电池除尘上料机构夹爪有OK料记忆
ANDNOT H86.02  ; RK_10 电池除尘上料机构夹爪有NG料记忆
AND H85.00  ; RK_10 U8_U 电池除尘上料X轴回原点记忆
LD 866.04  ; RK_10 U8_U 电池除尘上料X轴Hipot NG放料位标志
AND H87.00  ; RK_10 Hipot检测NG拉带放料位有料记忆
AND 818.07  ; RK_10 Hipot检测NG拉带有料感应#1标志[0018.07]
AND 818.08  ; RK_10 Hipot检测NG拉带有料感应#2标志[0018.08]
LD 866.03  ; RK_10 U8_U 电池除尘上料X轴Hipot OK放料位标志
AND H91.00  ; RK_11 电池除尘机构有料记忆
AND 811.04  ; RK_11 电池除尘有料感应标志[0011.04]
ORLD
ANDLD
ORLD
LD D1206.09  ; RK_10 电池除尘上料机构升降气缸上升（步）
AND 816.03  ; RK_10 电池除尘上料机械手升降气缸上升位标志[0016.03]
ORLD
LD D1206.10  ; RK_10 电池除尘上料机构#1/2Hipot检测取料位（步）
LDNOT W279.04  ; #1Hipot检测取料位有取电池需求
ANDNOT W279.05  ; #2Hipot检测取料位有取电池需求
OR W279.04  ; #1Hipot检测取料位有取电池需求
AND 866.01  ; RK_10 U8_U 电池除尘上料X轴#1Hipot检测取料位标志
LD W279.05  ; #2Hipot检测取料位有取电池需求
AND 866.02  ; RK_10 U8_U 电池除尘上料X轴#2Hipot检测取料位标志
ORLD
ANDLD
AND H85.00  ; RK_10 U8_U 电池除尘上料X轴回原点记忆
ORLD
OR D1206.11  ; 备用
LD D1204.01  ; RK_10 电池除尘上料机构单步/自动循环运行中
AND W1.01  ; 自动模式
@LD D1203.15  ; RK_10 电池除尘上料机构单步（SW）
AND D1204.10  ; RK_10 电池除尘上料机构单步运行条件
ORLD
ANDLD
OUT D1205.01  ; RK_10 电池除尘上料机构步进条件

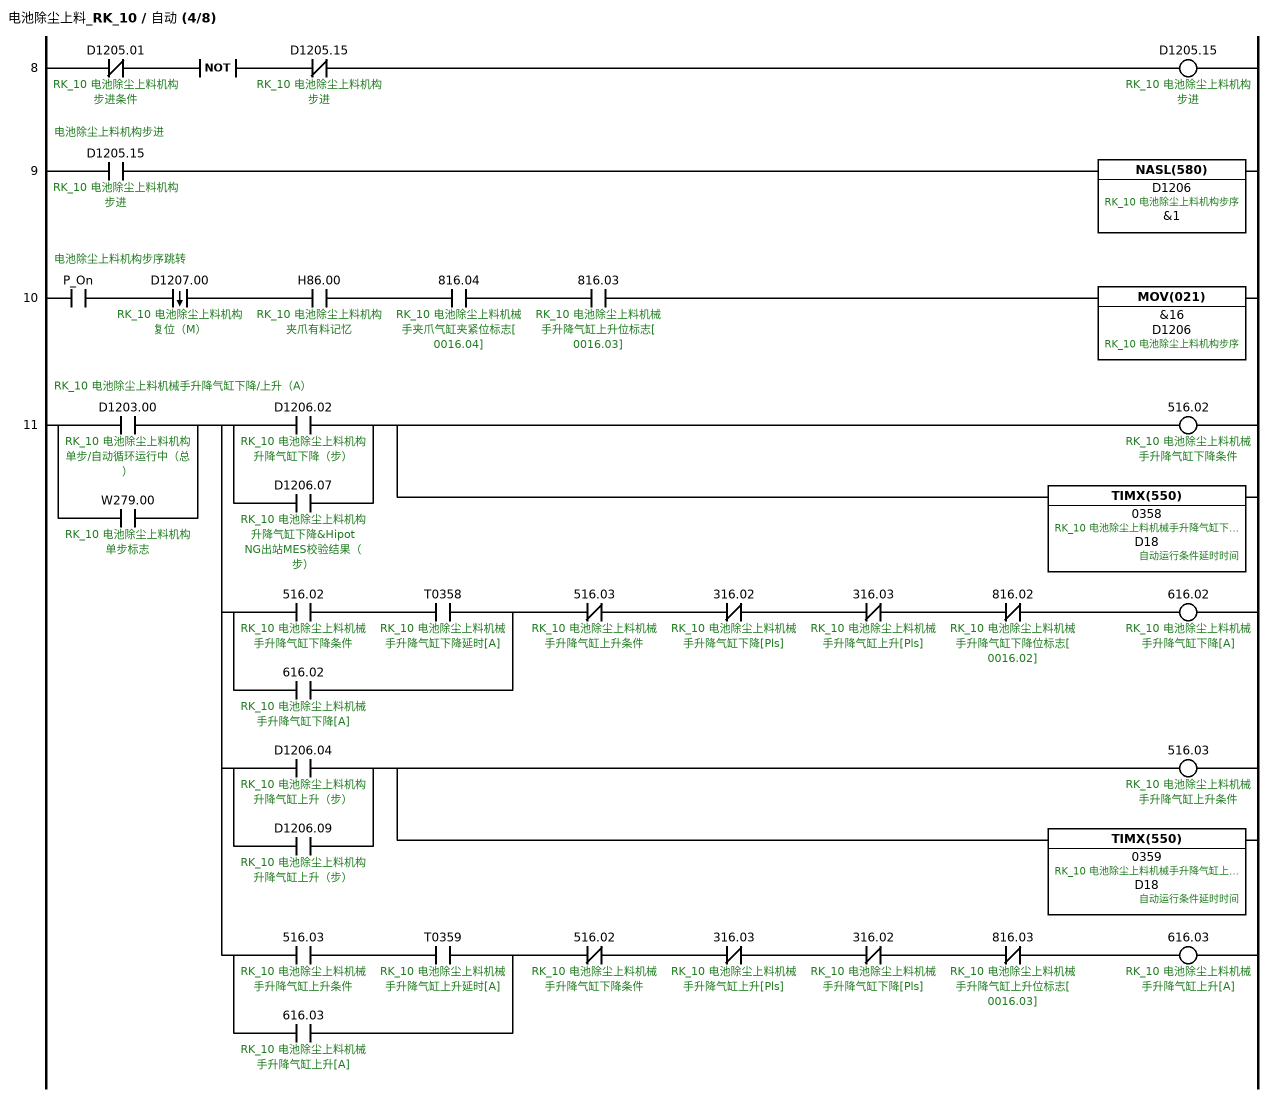
; rung 8
LDNOT D1205.01  ; RK_10 电池除尘上料机构步进条件
NOT(520)
ANDNOT D1205.15  ; RK_10 电池除尘上料机构步进
OUT D1205.15  ; RK_10 电池除尘上料机构步进
; rung 9: 电池除尘上料机构步进
LD D1205.15  ; RK_10 电池除尘上料机构步进
NASL(580) D1206 &1  ; RK_10 电池除尘上料机构步序
; rung 10: 电池除尘上料机构步序跳转
LD P_On
%AND D1207.00  ; RK_10 电池除尘上料机构复位（M）
AND H86.00  ; RK_10 电池除尘上料机构夹爪有料记忆
AND 816.04  ; RK_10 电池除尘上料机械手夹爪气缸夹紧位标志[0016.04]
AND 816.03  ; RK_10 电池除尘上料机械手升降气缸上升位标志[0016.03]
MOV(021) &16 D1206  ; RK_10 电池除尘上料机构步序  // RK_10 电池除尘上料机构升降气缸上升步（D1206.04）
; rung 11: RK_10 电池除尘上料机械手升降气缸下降/上升（A）
LD D1203.00  ; RK_10 电池除尘上料机构单步/自动循环运行中（总）
OR W279.00  ; RK_10 电池除尘上料机构单步标志
OUT TR0
LD D1206.02  ; RK_10 电池除尘上料机构升降气缸下降（步）
OR D1206.07  ; RK_10 电池除尘上料机构升降气缸下降&Hipot NG出站MES校验结果（步）
ANDLD
OUT 516.02  ; RK_10 电池除尘上料机械手升降气缸下降条件
TIMX(550) 0358 D18  ; 自动运行条件延时时间, RK_10 电池除尘上料机械手升降气缸下降延时[A]
LD TR0
LD 516.02  ; RK_10 电池除尘上料机械手升降气缸下降条件
AND T0358  ; RK_10 电池除尘上料机械手升降气缸下降延时[A]
OR 616.02  ; RK_10 电池除尘上料机械手升降气缸下降[A]
ANDLD
ANDNOT 516.03  ; RK_10 电池除尘上料机械手升降气缸上升条件
ANDNOT 316.02  ; RK_10 电池除尘上料机械手升降气缸下降[Pls]
ANDNOT 316.03  ; RK_10 电池除尘上料机械手升降气缸上升[Pls]
ANDNOT 816.02  ; RK_10 电池除尘上料机械手升降气缸下降位标志[0016.02]
OUT 616.02  ; RK_10 电池除尘上料机械手升降气缸下降[A]
LD TR0
LD D1206.04  ; RK_10 电池除尘上料机构升降气缸上升（步）
OR D1206.09  ; RK_10 电池除尘上料机构升降气缸上升（步）
ANDLD
OUT 516.03  ; RK_10 电池除尘上料机械手升降气缸上升条件
TIMX(550) 0359 D18  ; 自动运行条件延时时间, RK_10 电池除尘上料机械手升降气缸上升延时[A]
LD TR0
LD 516.03  ; RK_10 电池除尘上料机械手升降气缸上升条件
AND T0359  ; RK_10 电池除尘上料机械手升降气缸上升延时[A]
OR 616.03  ; RK_10 电池除尘上料机械手升降气缸上升[A]
ANDLD
ANDNOT 516.02  ; RK_10 电池除尘上料机械手升降气缸下降条件
ANDNOT 316.03  ; RK_10 电池除尘上料机械手升降气缸上升[Pls]
ANDNOT 316.02  ; RK_10 电池除尘上料机械手升降气缸下降[Pls]
ANDNOT 816.03  ; RK_10 电池除尘上料机械手升降气缸上升位标志[0016.03]
OUT 616.03  ; RK_10 电池除尘上料机械手升降气缸上升[A]

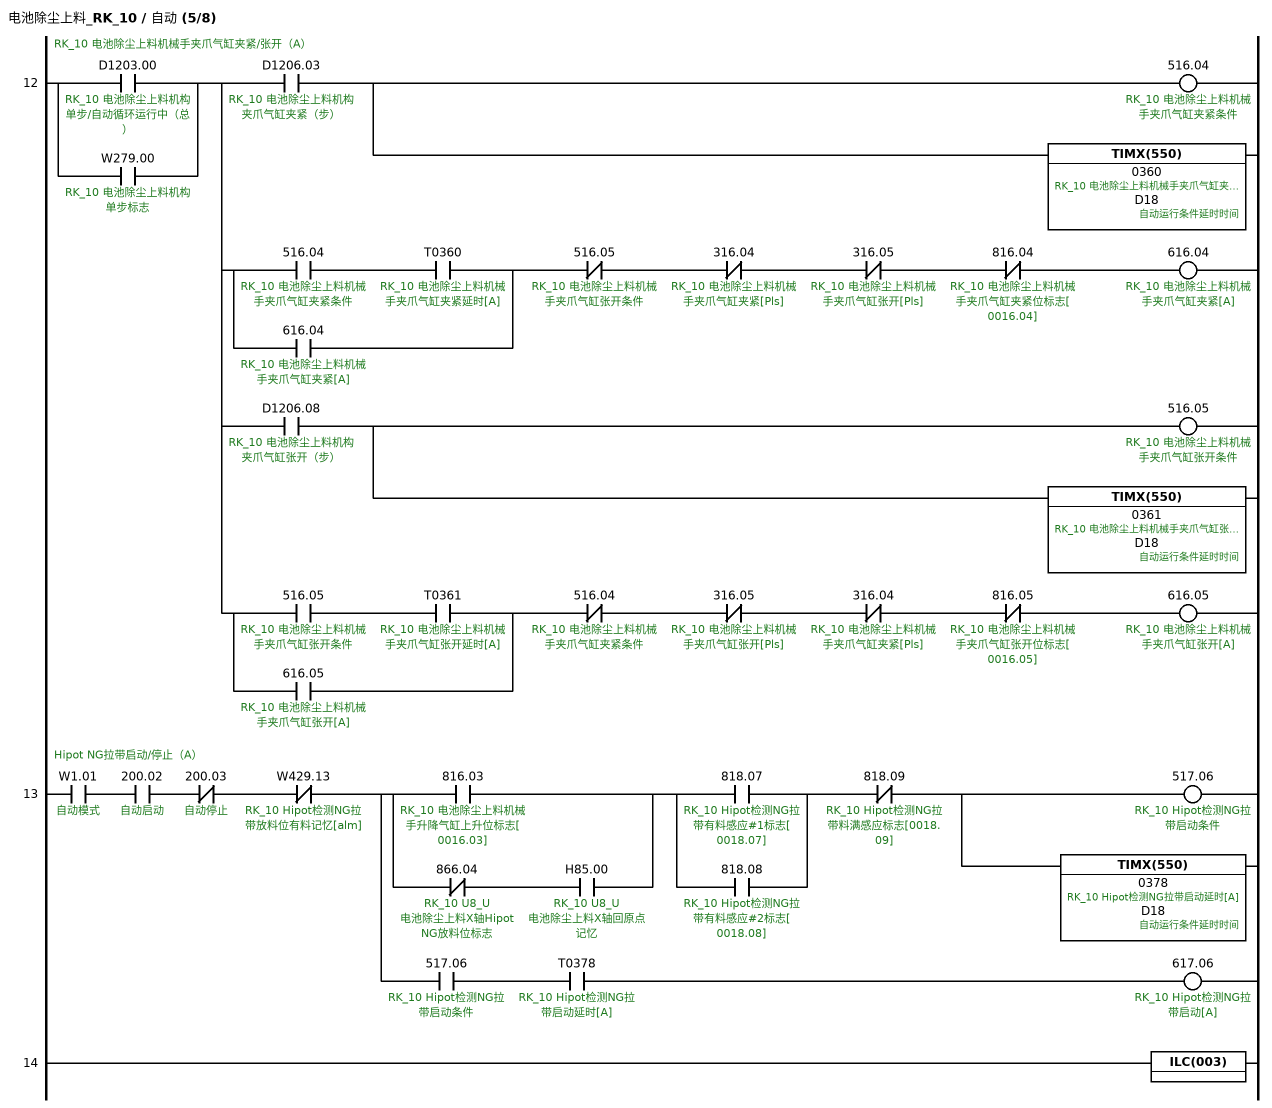
; rung 12: RK_10 电池除尘上料机械手夹爪气缸夹紧/张开（A）
LD D1203.00  ; RK_10 电池除尘上料机构单步/自动循环运行中（总）
OR W279.00  ; RK_10 电池除尘上料机构单步标志
OUT TR0
AND D1206.03  ; RK_10 电池除尘上料机构夹爪气缸夹紧（步）
OUT 516.04  ; RK_10 电池除尘上料机械手夹爪气缸夹紧条件
TIMX(550) 0360 D18  ; 自动运行条件延时时间, RK_10 电池除尘上料机械手夹爪气缸夹紧延时[A]
LD TR0
LD 516.04  ; RK_10 电池除尘上料机械手夹爪气缸夹紧条件
AND T0360  ; RK_10 电池除尘上料机械手夹爪气缸夹紧延时[A]
OR 616.04  ; RK_10 电池除尘上料机械手夹爪气缸夹紧[A]
ANDLD
ANDNOT 516.05  ; RK_10 电池除尘上料机械手夹爪气缸张开条件
ANDNOT 316.04  ; RK_10 电池除尘上料机械手夹爪气缸夹紧[Pls]
ANDNOT 316.05  ; RK_10 电池除尘上料机械手夹爪气缸张开[Pls]
ANDNOT 816.04  ; RK_10 电池除尘上料机械手夹爪气缸夹紧位标志[0016.04]
OUT 616.04  ; RK_10 电池除尘上料机械手夹爪气缸夹紧[A]
LD TR0
AND D1206.08  ; RK_10 电池除尘上料机构夹爪气缸张开（步）
OUT 516.05  ; RK_10 电池除尘上料机械手夹爪气缸张开条件
TIMX(550) 0361 D18  ; 自动运行条件延时时间, RK_10 电池除尘上料机械手夹爪气缸张开延时[A]
LD TR0
LD 516.05  ; RK_10 电池除尘上料机械手夹爪气缸张开条件
AND T0361  ; RK_10 电池除尘上料机械手夹爪气缸张开延时[A]
OR 616.05  ; RK_10 电池除尘上料机械手夹爪气缸张开[A]
ANDLD
ANDNOT 516.04  ; RK_10 电池除尘上料机械手夹爪气缸夹紧条件
ANDNOT 316.05  ; RK_10 电池除尘上料机械手夹爪气缸张开[Pls]
ANDNOT 316.04  ; RK_10 电池除尘上料机械手夹爪气缸夹紧[Pls]
ANDNOT 816.05  ; RK_10 电池除尘上料机械手夹爪气缸张开位标志[0016.05]
OUT 616.05  ; RK_10 电池除尘上料机械手夹爪气缸张开[A]
; rung 13: Hipot NG拉带启动/停止（A）
LD W1.01  ; 自动模式
AND 200.02  ; 自动启动
ANDNOT 200.03  ; 自动停止
ANDNOT W429.13  ; RK_10 Hipot检测NG拉带放料位有料记忆[alm]
OUT TR0
LD 816.03  ; RK_10 电池除尘上料机械手升降气缸上升位标志[0016.03]
LDNOT 866.04  ; RK_10 U8_U 电池除尘上料X轴Hipot NG放料位标志
AND H85.00  ; RK_10 U8_U 电池除尘上料X轴回原点记忆
ORLD
ANDLD
LD 818.07  ; RK_10 Hipot检测NG拉带有料感应#1标志[0018.07]
OR 818.08  ; RK_10 Hipot检测NG拉带有料感应#2标志[0018.08]
ANDLD
ANDNOT 818.09  ; RK_10 Hipot检测NG拉带料满感应标志[0018.09]
OUT 517.06  ; RK_10 Hipot检测NG拉带启动条件
TIMX(550) 0378 D18  ; 自动运行条件延时时间, RK_10 Hipot检测NG拉带启动延时[A]
LD TR0
AND 517.06  ; RK_10 Hipot检测NG拉带启动条件
AND T0378  ; RK_10 Hipot检测NG拉带启动延时[A]
OUT 617.06  ; RK_10 Hipot检测NG拉带启动[A]
; rung 14
ILC(003)

